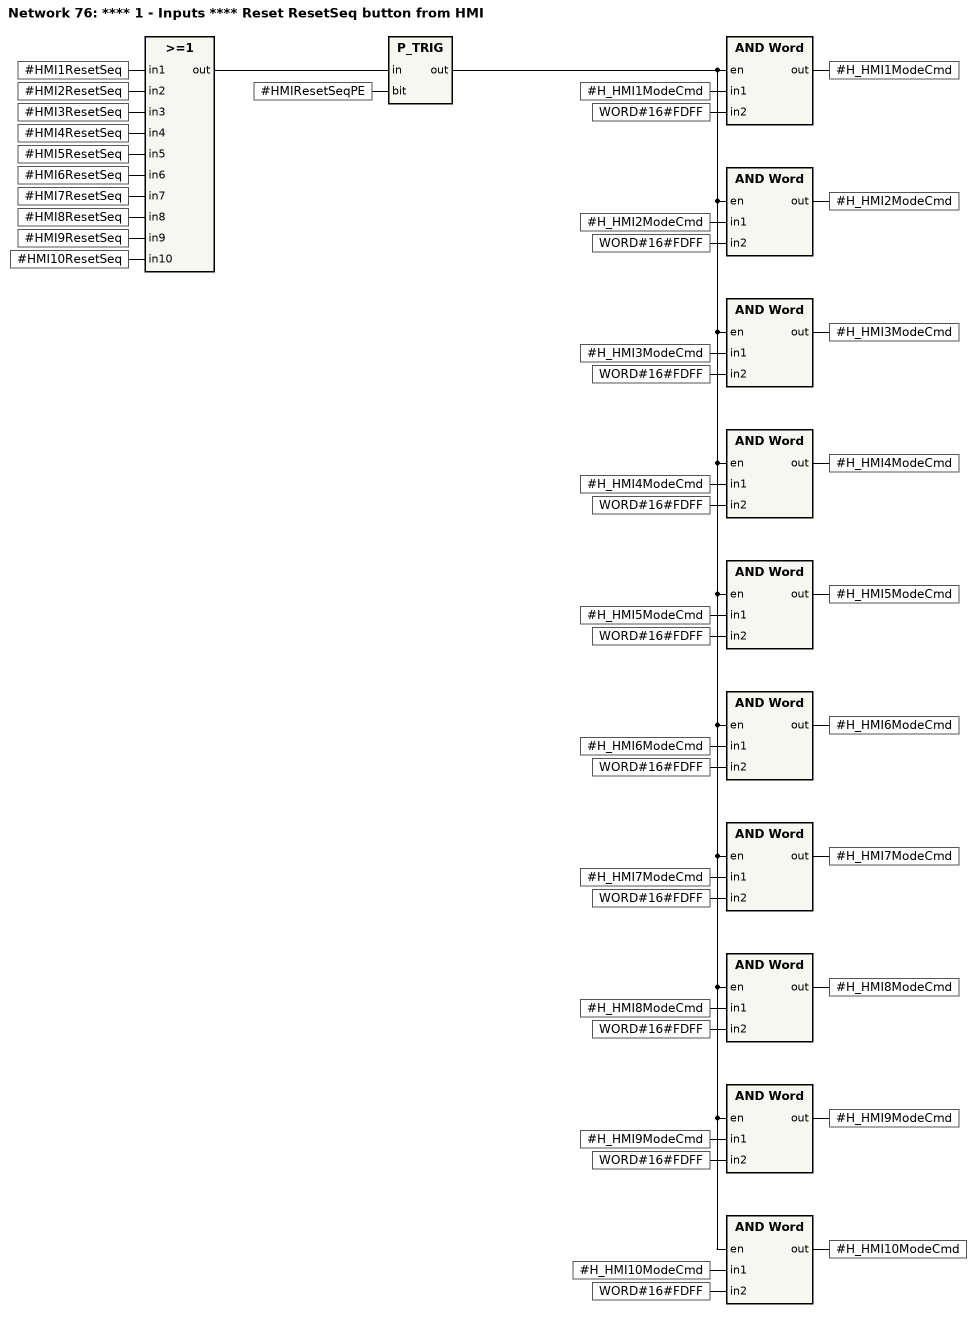
   #_w1 := #HMI1ResetSeq OR #HMI2ResetSeq OR #HMI3ResetSeq OR #HMI4ResetSeq OR #HMI5ResetSeq OR #HMI6ResetSeq OR #HMI7ResetSeq OR #HMI8ResetSeq OR #HMI9ResetSeq OR #HMI10ResetSeq;
   #_w2 := #_w1 AND NOT #HMIResetSeqPE;   // rising edge
   #HMIResetSeqPE := #_w1;
   IF #_w2 THEN
       #H_HMI1ModeCmd := #H_HMI1ModeCmd AND WORD#16#FDFF;
       #H_HMI2ModeCmd := #H_HMI2ModeCmd AND WORD#16#FDFF;
       #H_HMI3ModeCmd := #H_HMI3ModeCmd AND WORD#16#FDFF;
       #H_HMI4ModeCmd := #H_HMI4ModeCmd AND WORD#16#FDFF;
       #H_HMI5ModeCmd := #H_HMI5ModeCmd AND WORD#16#FDFF;
       #H_HMI6ModeCmd := #H_HMI6ModeCmd AND WORD#16#FDFF;
       #H_HMI7ModeCmd := #H_HMI7ModeCmd AND WORD#16#FDFF;
       #H_HMI8ModeCmd := #H_HMI8ModeCmd AND WORD#16#FDFF;
       #H_HMI9ModeCmd := #H_HMI9ModeCmd AND WORD#16#FDFF;
       #H_HMI10ModeCmd := #H_HMI10ModeCmd AND WORD#16#FDFF;
   END_IF;
END_REGION

REGION Network 77: **** 1 - Inputs **** Reset LockManual button from HMI
   // Reset LockManual button from HMI
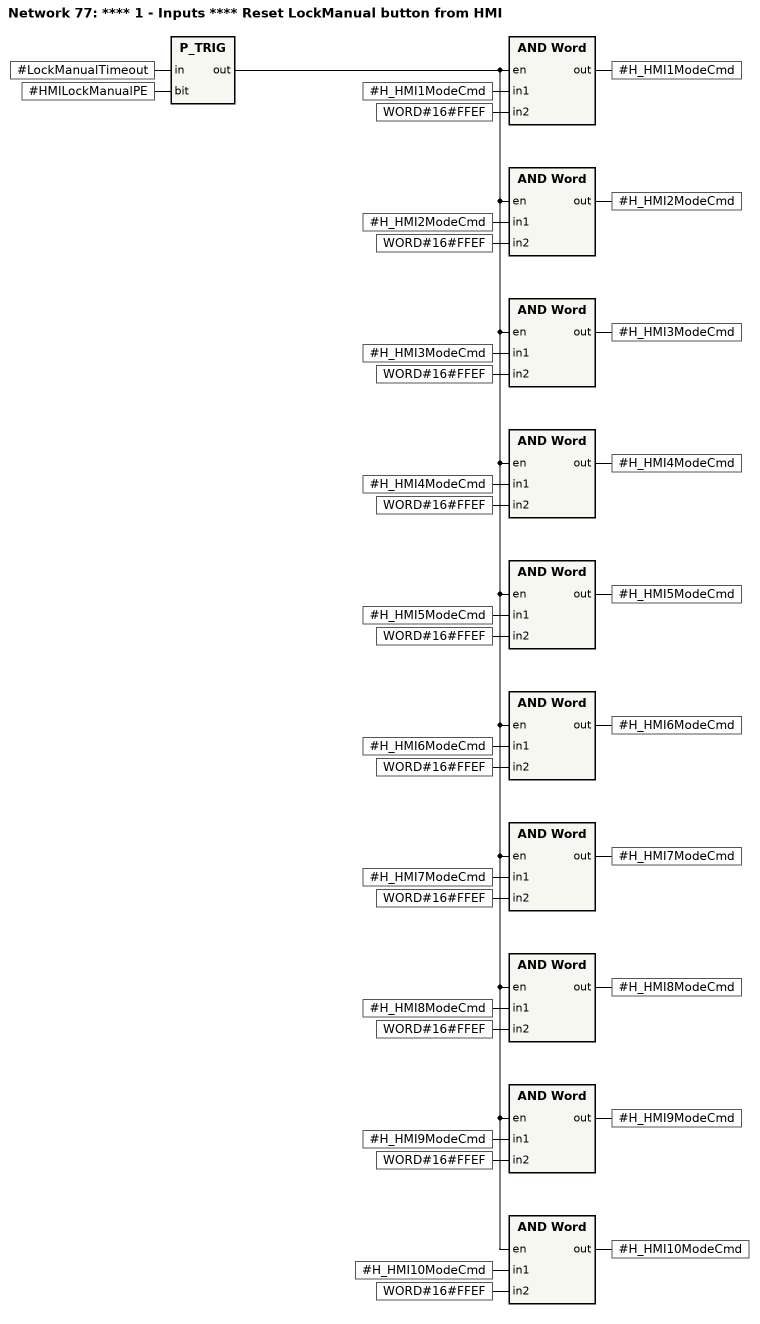
   #_w1 := #LockManualTimeout AND NOT #HMILockManualPE;   // rising edge
   #HMILockManualPE := #LockManualTimeout;
   IF #_w1 THEN
       #H_HMI1ModeCmd := #H_HMI1ModeCmd AND WORD#16#FFEF;
       #H_HMI2ModeCmd := #H_HMI2ModeCmd AND WORD#16#FFEF;
       #H_HMI3ModeCmd := #H_HMI3ModeCmd AND WORD#16#FFEF;
       #H_HMI4ModeCmd := #H_HMI4ModeCmd AND WORD#16#FFEF;
       #H_HMI5ModeCmd := #H_HMI5ModeCmd AND WORD#16#FFEF;
       #H_HMI6ModeCmd := #H_HMI6ModeCmd AND WORD#16#FFEF;
       #H_HMI7ModeCmd := #H_HMI7ModeCmd AND WORD#16#FFEF;
       #H_HMI8ModeCmd := #H_HMI8ModeCmd AND WORD#16#FFEF;
       #H_HMI9ModeCmd := #H_HMI9ModeCmd AND WORD#16#FFEF;
       #H_HMI10ModeCmd := #H_HMI10ModeCmd AND WORD#16#FFEF;
   END_IF;
END_REGION

REGION Network 78: **** 1 - Inputs **** Set Auto select on HMI-1 if plc go from STOP to RUN
   // Set Auto select on HMI-1 with the first scan
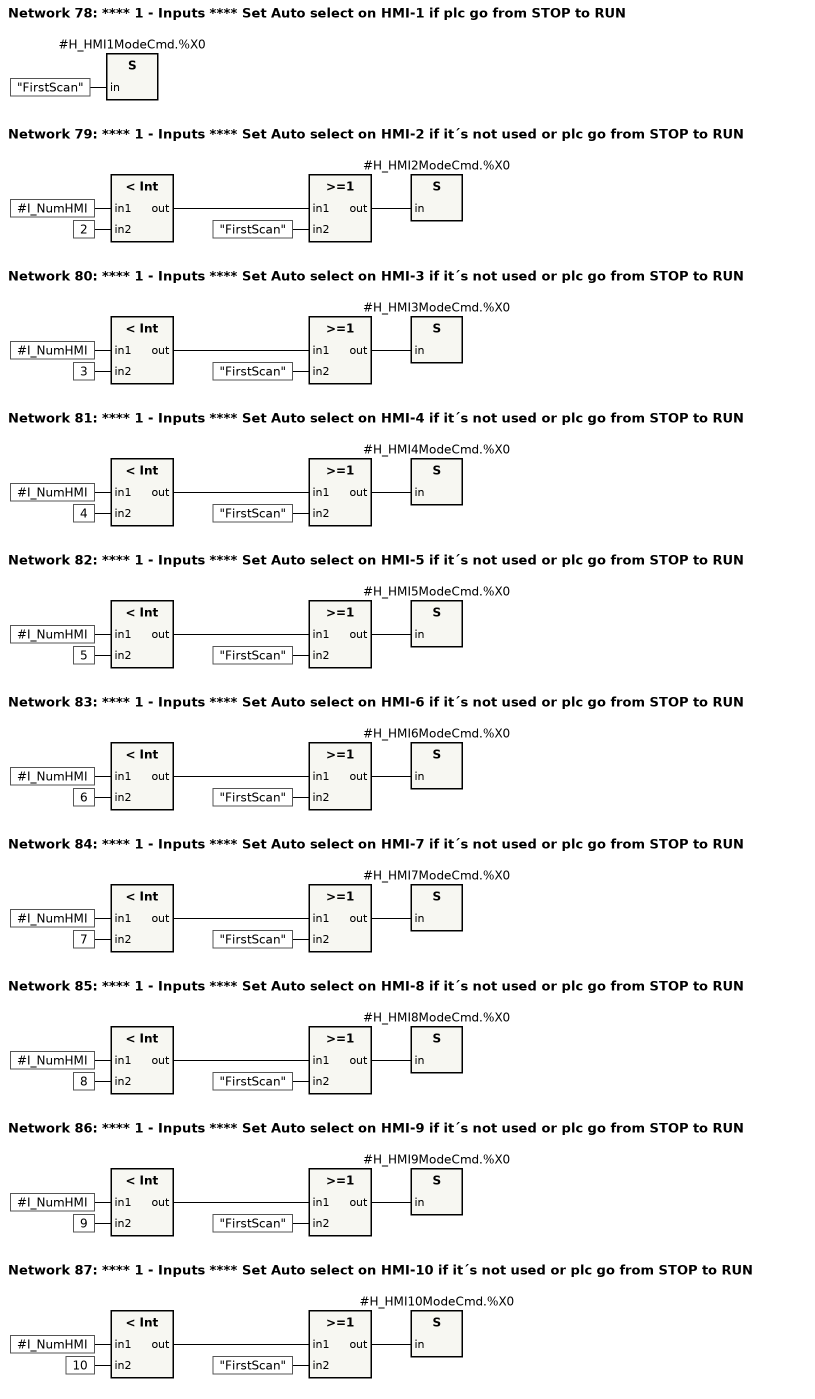
   IF "FirstScan" THEN #H_HMI1ModeCmd.%X0 := TRUE; END_IF;
END_REGION

REGION Network 79: **** 1 - Inputs **** Set Auto select on HMI-2 if it´s not used or plc go from STOP to RUN
   // Set Auto select on HMI-2 if it´s not used
   IF (#I_NumHMI < 2) OR "FirstScan" THEN #H_HMI2ModeCmd.%X0 := TRUE; END_IF;
END_REGION

REGION Network 80: **** 1 - Inputs **** Set Auto select on HMI-3 if it´s not used or plc go from STOP to RUN
   // Set Auto select on HMI-3 if it´s not used
   IF (#I_NumHMI < 3) OR "FirstScan" THEN #H_HMI3ModeCmd.%X0 := TRUE; END_IF;
END_REGION

REGION Network 81: **** 1 - Inputs **** Set Auto select on HMI-4 if it´s not used or plc go from STOP to RUN
   // Set Auto select on HMI-4 if it´s not used
   IF (#I_NumHMI < 4) OR "FirstScan" THEN #H_HMI4ModeCmd.%X0 := TRUE; END_IF;
END_REGION

REGION Network 82: **** 1 - Inputs **** Set Auto select on HMI-5 if it´s not used or plc go from STOP to RUN
   // Set Auto select on HMI-5 if it´s not used
   IF (#I_NumHMI < 5) OR "FirstScan" THEN #H_HMI5ModeCmd.%X0 := TRUE; END_IF;
END_REGION

REGION Network 83: **** 1 - Inputs **** Set Auto select on HMI-6 if it´s not used or plc go from STOP to RUN
   // Set Auto select on HMI-6 if it´s not used
   IF (#I_NumHMI < 6) OR "FirstScan" THEN #H_HMI6ModeCmd.%X0 := TRUE; END_IF;
END_REGION

REGION Network 84: **** 1 - Inputs **** Set Auto select on HMI-7 if it´s not used or plc go from STOP to RUN
   // Set Auto select on HMI-7 if it´s not used
   IF (#I_NumHMI < 7) OR "FirstScan" THEN #H_HMI7ModeCmd.%X0 := TRUE; END_IF;
END_REGION

REGION Network 85: **** 1 - Inputs **** Set Auto select on HMI-8 if it´s not used or plc go from STOP to RUN
   // Set Auto select on HMI-8 if it´s not used
   IF (#I_NumHMI < 8) OR "FirstScan" THEN #H_HMI8ModeCmd.%X0 := TRUE; END_IF;
END_REGION

REGION Network 86: **** 1 - Inputs **** Set Auto select on HMI-9 if it´s not used or plc go from STOP to RUN
   // Set Auto select on HMI-9 if it´s not used
   IF (#I_NumHMI < 9) OR "FirstScan" THEN #H_HMI9ModeCmd.%X0 := TRUE; END_IF;
END_REGION

REGION Network 87: **** 1 - Inputs **** Set Auto select on HMI-10 if it´s not used or plc go from STOP to RUN
   // Set Auto select on HMI-10 if it´s not used
   IF (#I_NumHMI < 10) OR "FirstScan" THEN #H_HMI10ModeCmd.%X0 := TRUE; END_IF;
END_REGION

REGION Network 88: **** 4.3 - Machine Status - Operator Sel **** Forced manual is selected on the active HMI
   // Forced manual is selected on the active HMI
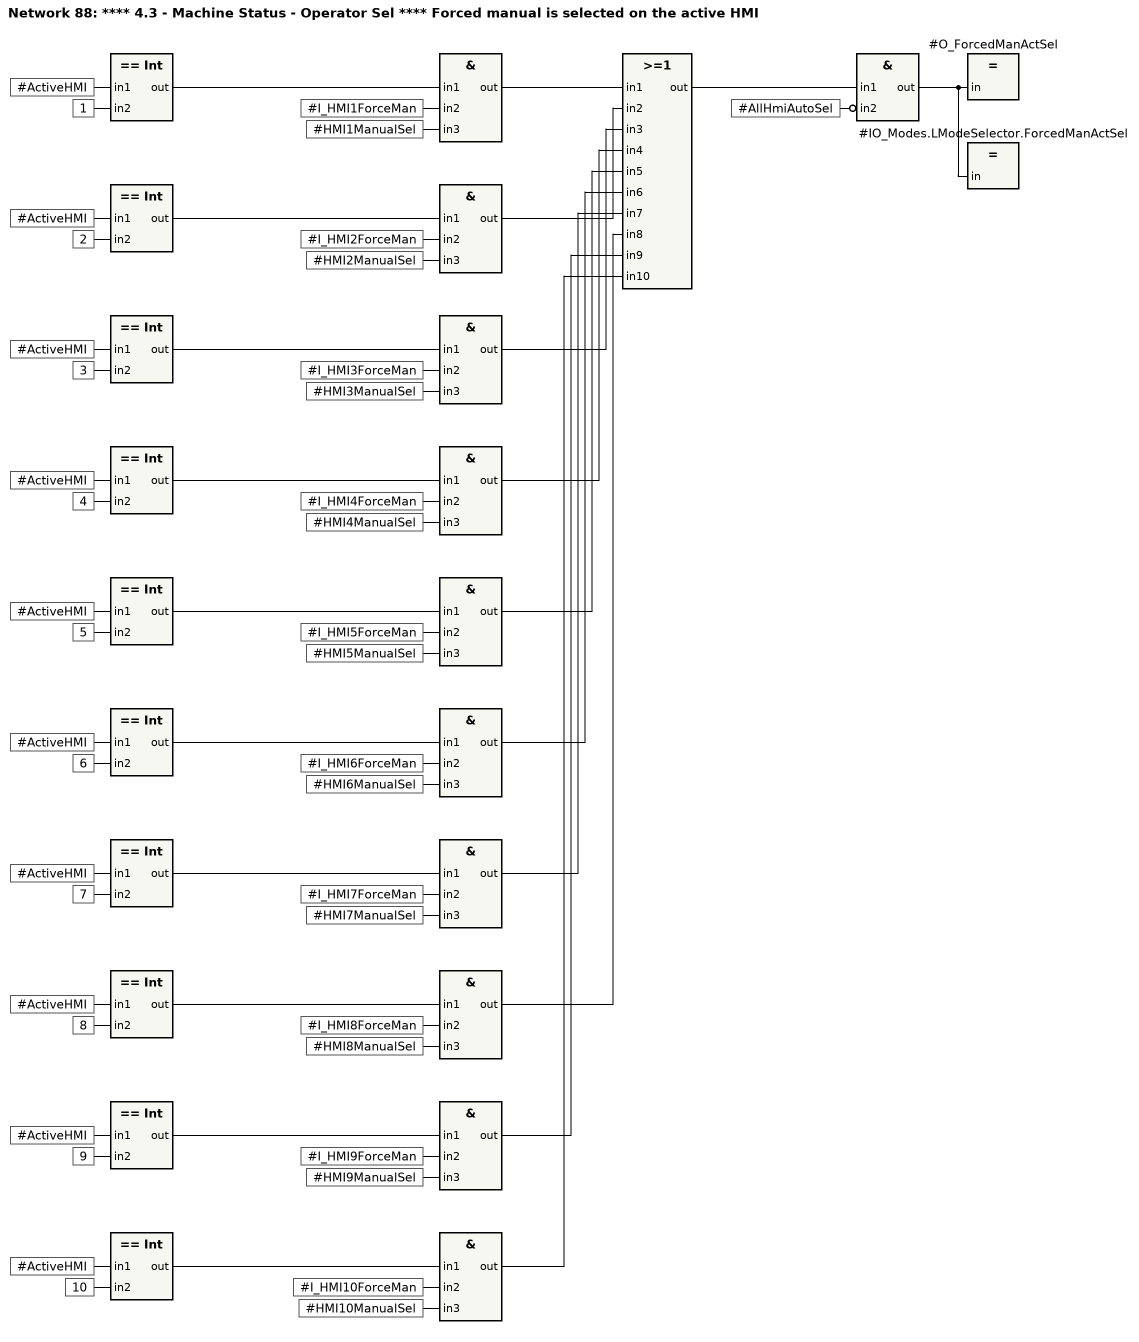
   #O_ForcedManActSel := (((#ActiveHMI = 1) AND #I_HMI1ForceMan AND #HMI1ManualSel) OR ((#ActiveHMI = 2) AND #I_HMI2ForceMan AND #HMI2ManualSel) OR ((#ActiveHMI = 3) AND #I_HMI3ForceMan AND #HMI3ManualSel) OR ((#ActiveHMI = 4) AND #I_HMI4ForceMan AND #HMI4ManualSel) OR ((#ActiveHMI = 5) AND #I_HMI5ForceMan AND #HMI5ManualSel) OR ((#ActiveHMI = 6) AND #I_HMI6ForceMan AND #HMI6ManualSel) OR ((#ActiveHMI = 7) AND #I_HMI7ForceMan AND #HMI7ManualSel) OR ((#ActiveHMI = 8) AND #I_HMI8ForceMan AND #HMI8ManualSel) OR ((#ActiveHMI = 9) AND #I_HMI9ForceMan AND #HMI9ManualSel) OR ((#ActiveHMI = 10) AND #I_HMI10ForceMan AND #HMI10ManualSel)) AND NOT #AllHmiAutoSel;
   #IO_Modes.LModeSelector.ForcedManActSel := #O_ForcedManActSel;
END_REGION

REGION Network 89: **** 4.3 - Machine Status - Operator Sel **** Set pushbutton is selected on the active HMI
   // Set pushbutton is selected on the active HMI
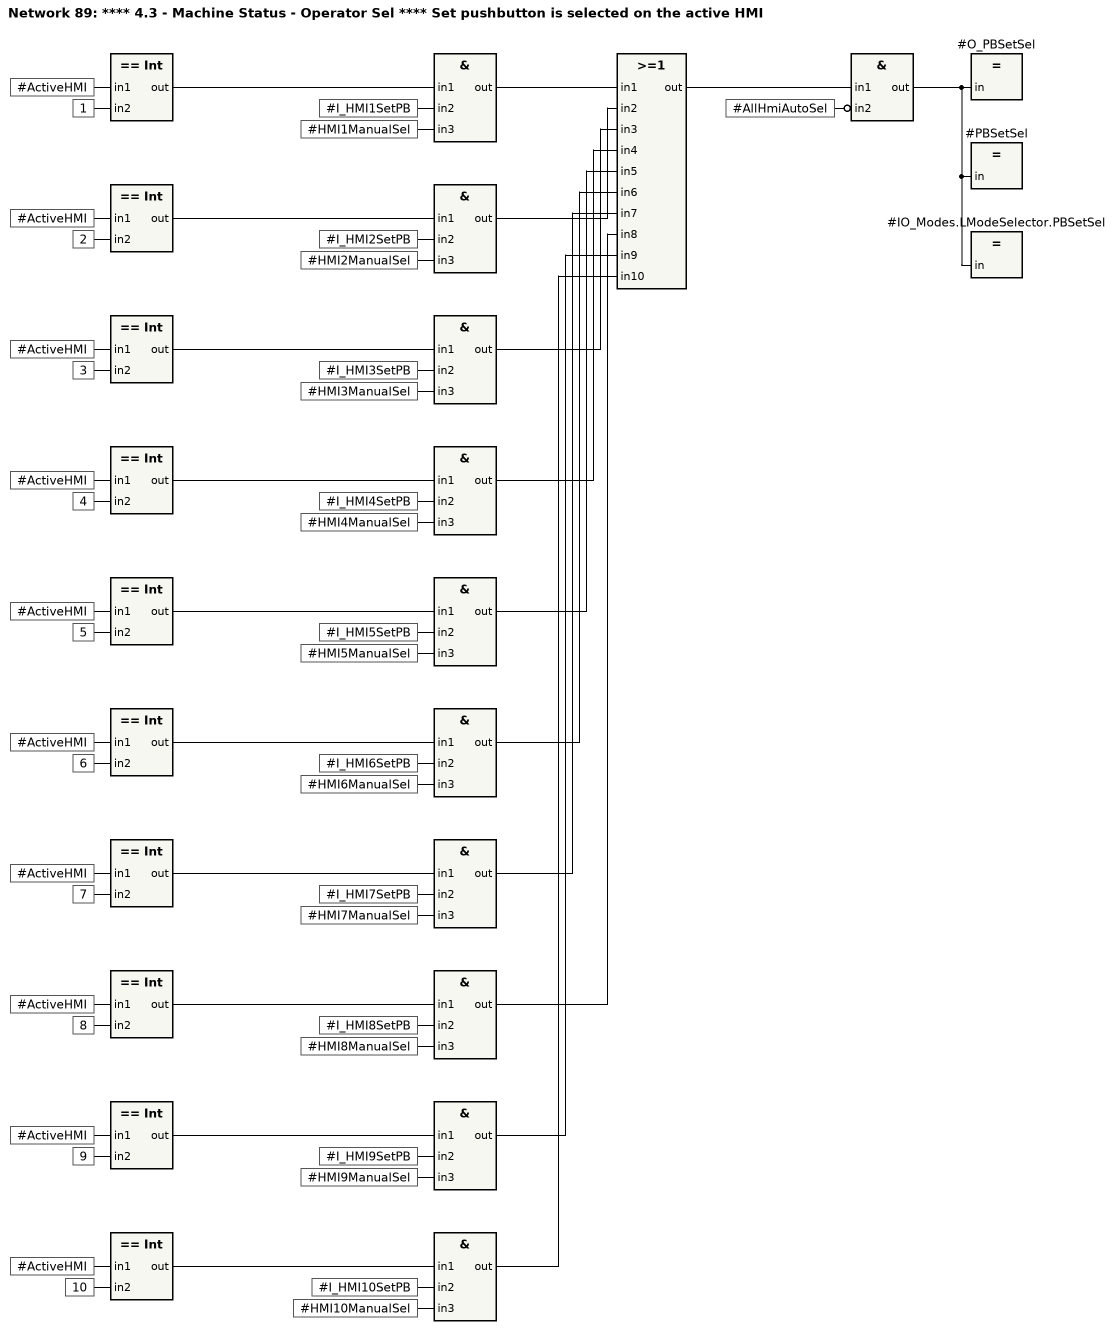
   #O_PBSetSel := (((#ActiveHMI = 1) AND #I_HMI1SetPB AND #HMI1ManualSel) OR ((#ActiveHMI = 2) AND #I_HMI2SetPB AND #HMI2ManualSel) OR ((#ActiveHMI = 3) AND #I_HMI3SetPB AND #HMI3ManualSel) OR ((#ActiveHMI = 4) AND #I_HMI4SetPB AND #HMI4ManualSel) OR ((#ActiveHMI = 5) AND #I_HMI5SetPB AND #HMI5ManualSel) OR ((#ActiveHMI = 6) AND #I_HMI6SetPB AND #HMI6ManualSel) OR ((#ActiveHMI = 7) AND #I_HMI7SetPB AND #HMI7ManualSel) OR ((#ActiveHMI = 8) AND #I_HMI8SetPB AND #HMI8ManualSel) OR ((#ActiveHMI = 9) AND #I_HMI9SetPB AND #HMI9ManualSel) OR ((#ActiveHMI = 10) AND #I_HMI10SetPB AND #HMI10ManualSel)) AND NOT #AllHmiAutoSel;
   #PBSetSel := #O_PBSetSel;
   #IO_Modes.LModeSelector.PBSetSel := #O_PBSetSel;
END_REGION

REGION Network 90: **** 4.3 - Machine Status - Operator Sel **** Reset pushbutton is selected on the active HMI
   // Reset pushbutton is selected on the active HMI
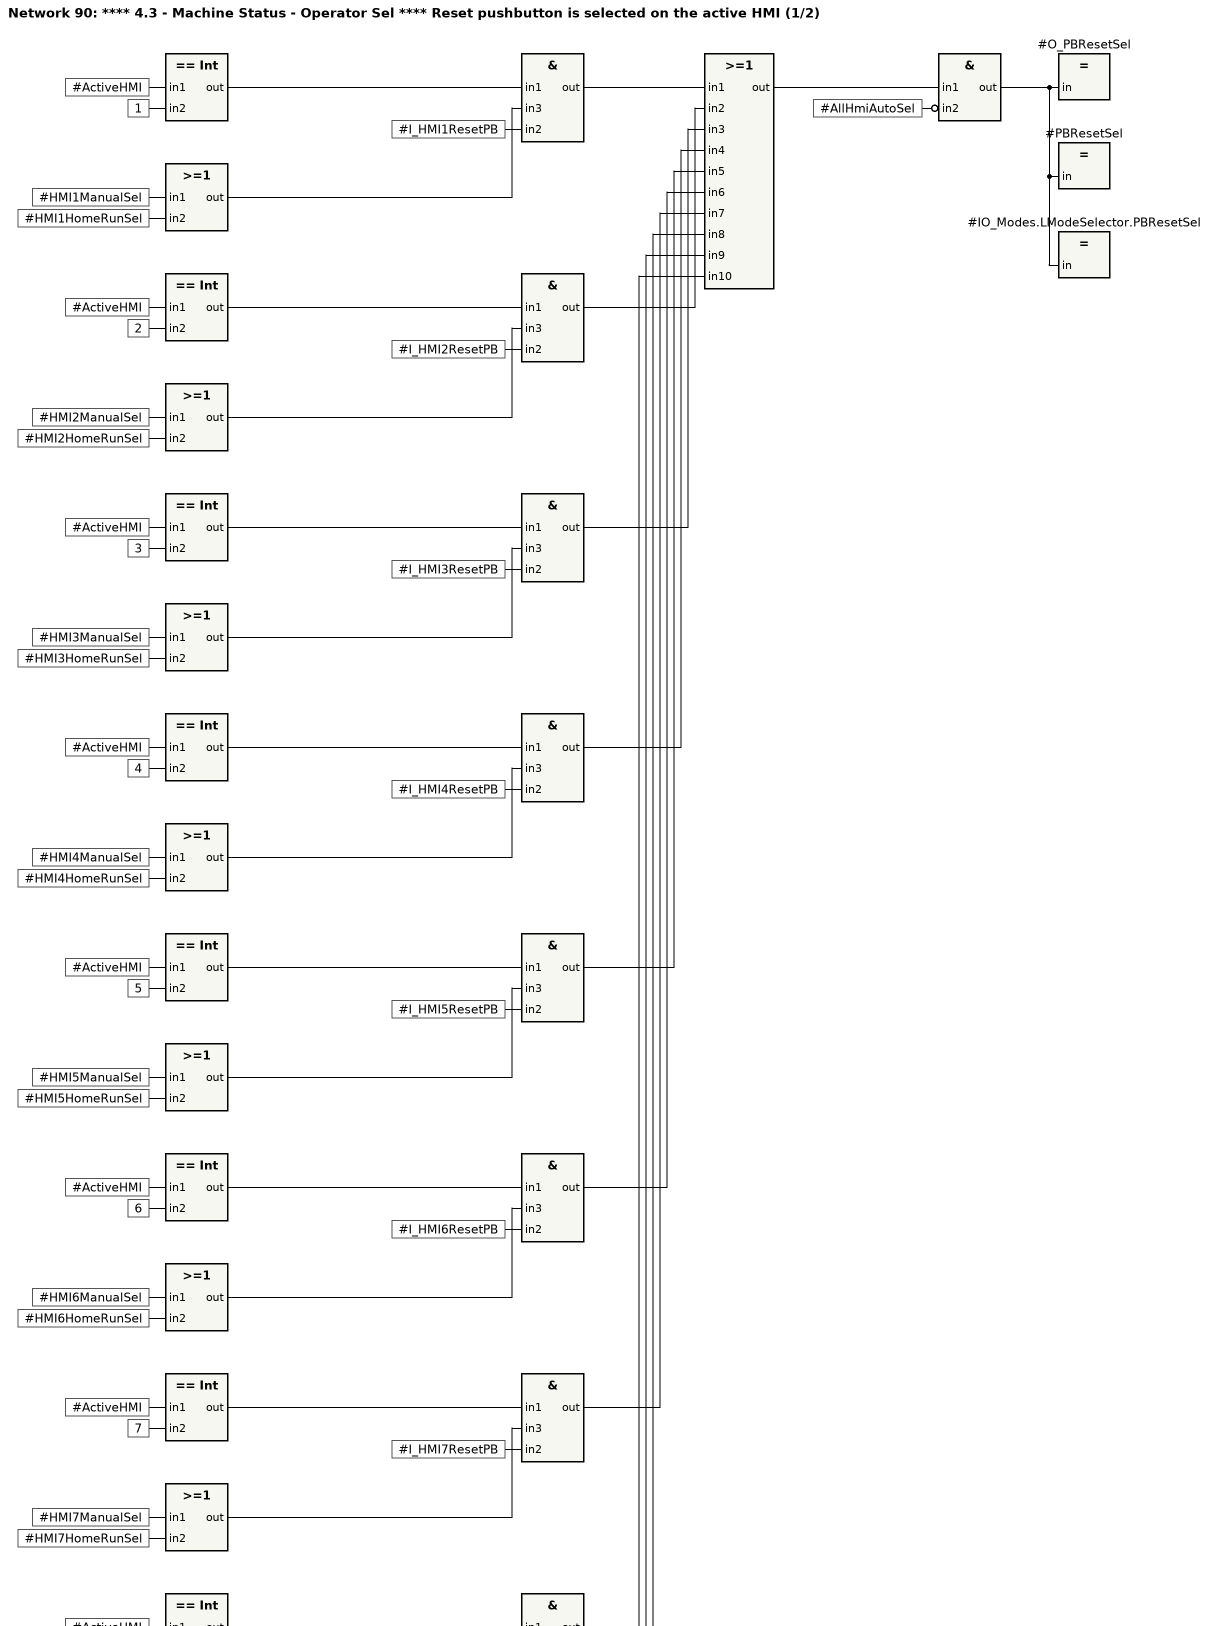
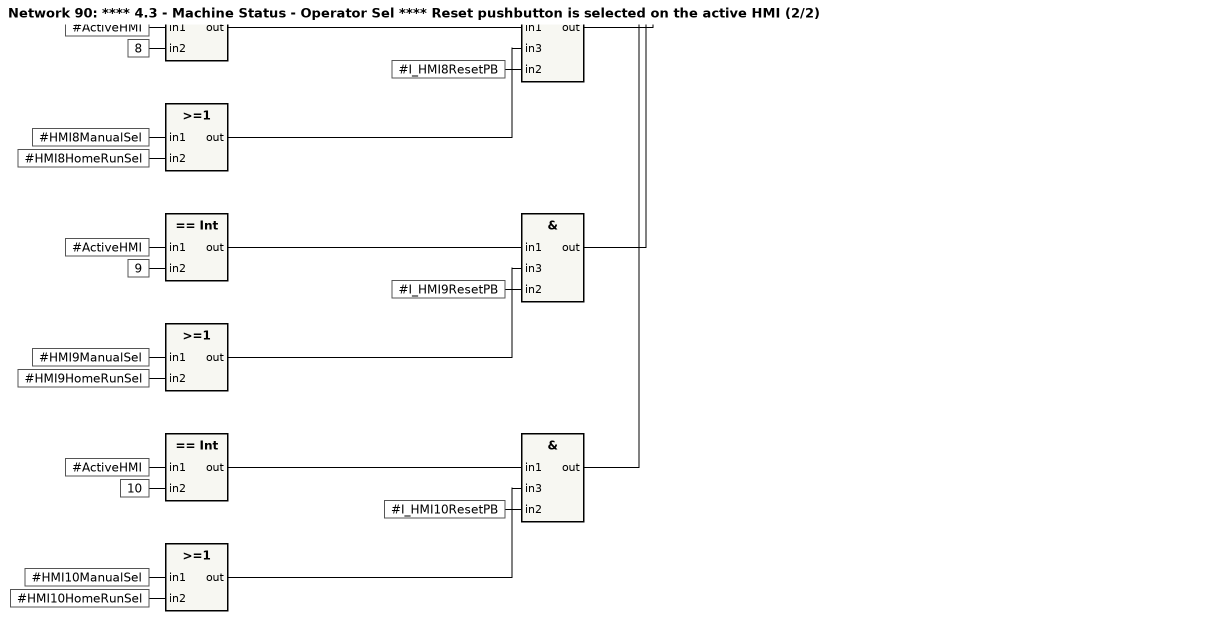
   #O_PBResetSel := (((#ActiveHMI = 1) AND (#HMI1ManualSel OR #HMI1HomeRunSel) AND #I_HMI1ResetPB) OR ((#ActiveHMI = 2) AND (#HMI2ManualSel OR #HMI2HomeRunSel) AND #I_HMI2ResetPB) OR ((#ActiveHMI = 3) AND (#HMI3ManualSel OR #HMI3HomeRunSel) AND #I_HMI3ResetPB) OR ((#ActiveHMI = 4) AND (#HMI4ManualSel OR #HMI4HomeRunSel) AND #I_HMI4ResetPB) OR ((#ActiveHMI = 5) AND (#HMI5ManualSel OR #HMI5HomeRunSel) AND #I_HMI5ResetPB) OR ((#ActiveHMI = 6) AND (#HMI6ManualSel OR #HMI6HomeRunSel) AND #I_HMI6ResetPB) OR ((#ActiveHMI = 7) AND (#HMI7ManualSel OR #HMI7HomeRunSel) AND #I_HMI7ResetPB) OR ((#ActiveHMI = 8) AND (#HMI8ManualSel OR #HMI8HomeRunSel) AND #I_HMI8ResetPB) OR ((#ActiveHMI = 9) AND (#HMI9ManualSel OR #HMI9HomeRunSel) AND #I_HMI9ResetPB) OR ((#ActiveHMI = 10) AND (#HMI10ManualSel OR #HMI10HomeRunSel) AND #I_HMI10ResetPB)) AND NOT #AllHmiAutoSel;
   #PBResetSel := #O_PBResetSel;
   #IO_Modes.LModeSelector.PBResetSel := #O_PBResetSel;
END_REGION

REGION Network 91: **** 4.3 - Machine Status - Operator Sel **** Homerun Redo is selected
   // Homerun Redo is selected
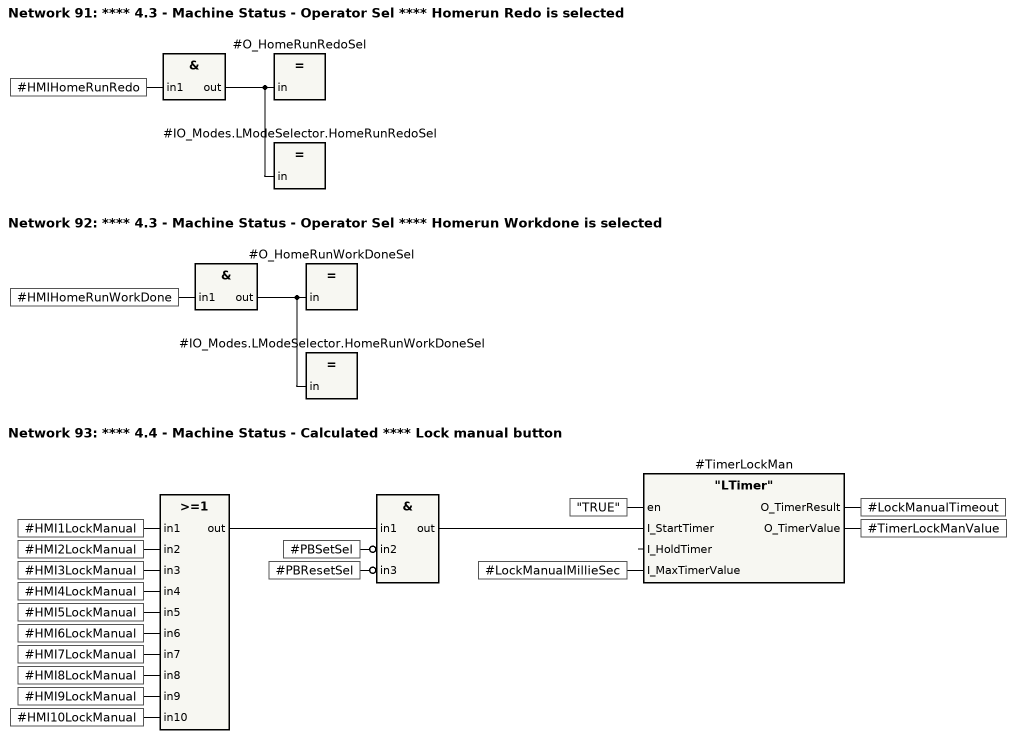
   #O_HomeRunRedoSel := #HMIHomeRunRedo;
   #IO_Modes.LModeSelector.HomeRunRedoSel := #HMIHomeRunRedo;
END_REGION

REGION Network 92: **** 4.3 - Machine Status - Operator Sel **** Homerun Workdone is selected
   // Homerun Workdone is selected
   #O_HomeRunWorkDoneSel := #HMIHomeRunWorkDone;
   #IO_Modes.LModeSelector.HomeRunWorkDoneSel := #HMIHomeRunWorkDone;
END_REGION

REGION Network 93: **** 4.4 - Machine Status - Calculated **** Lock manual button
   // Lock manual button
   IF "TRUE" THEN
       #TimerLockMan(I_StartTimer := (#HMI1LockManual OR #HMI2LockManual OR #HMI3LockManual OR #HMI4LockManual OR #HMI5LockManual OR #HMI6LockManual OR #HMI7LockManual OR #HMI8LockManual OR #HMI9LockManual OR #HMI10LockManual) AND NOT #PBSetSel AND NOT #PBResetSel,   // "LTimer"
                     I_MaxTimerValue := #LockManualMillieSec,
                     O_TimerResult => #LockManualTimeout,
                     O_TimerValue => #TimerLockManValue);
   END_IF;
END_REGION

REGION Network 94: **** 4.5 - Machine Status - Modes **** Auto is selected on all HMI
   // Auto is selected on all HMI
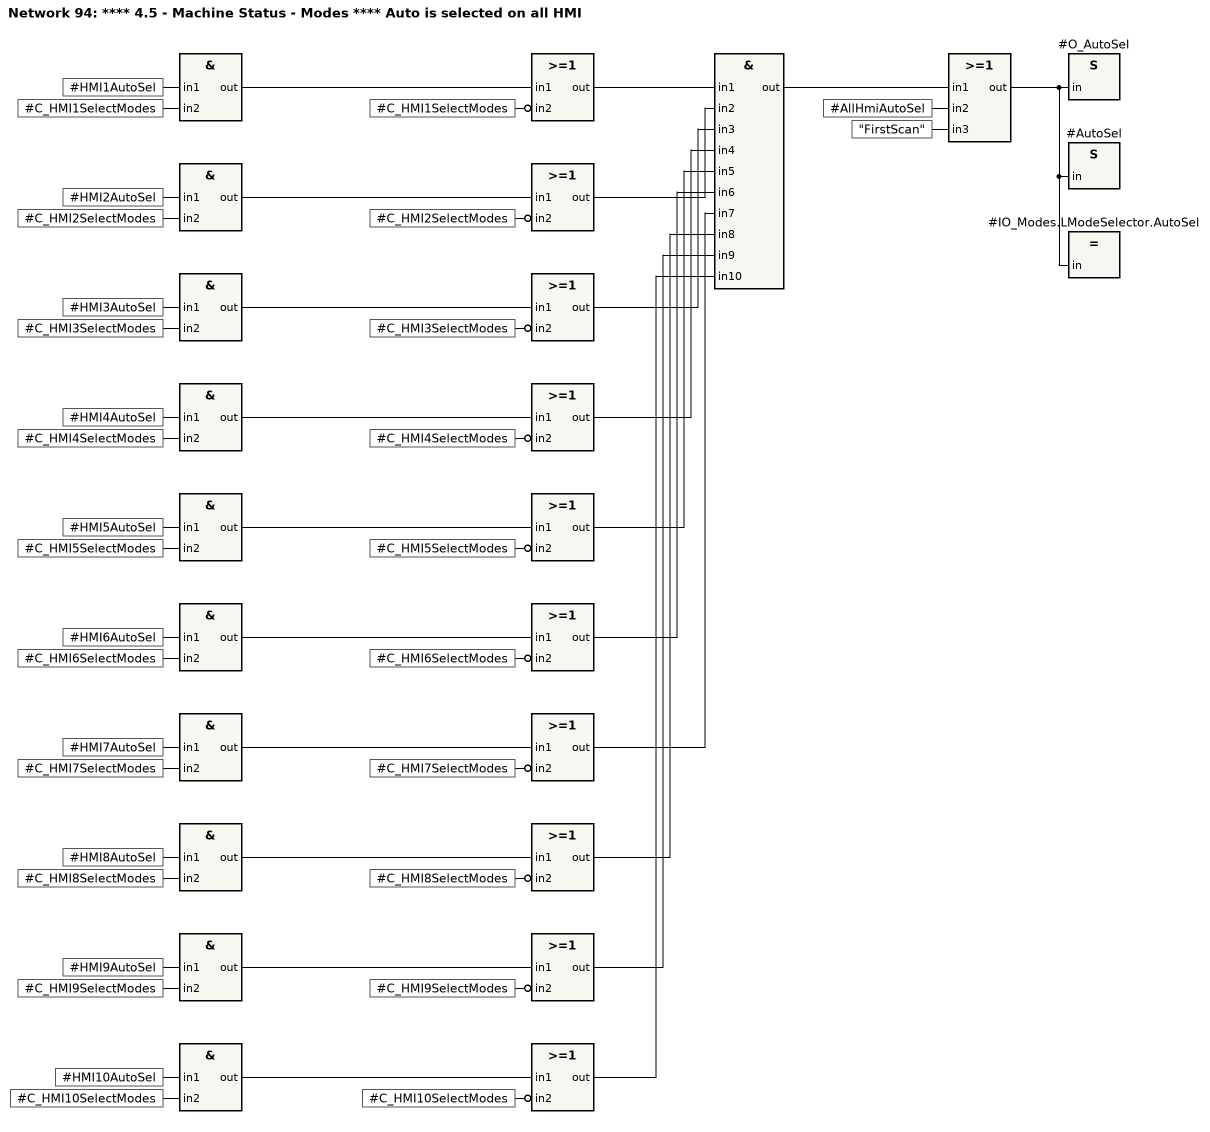
   #_w1 := (((#HMI1AutoSel AND #C_HMI1SelectModes) OR NOT #C_HMI1SelectModes) AND ((#HMI2AutoSel AND #C_HMI2SelectModes) OR NOT #C_HMI2SelectModes) AND ((#HMI3AutoSel AND #C_HMI3SelectModes) OR NOT #C_HMI3SelectModes) AND ((#HMI4AutoSel AND #C_HMI4SelectModes) OR NOT #C_HMI4SelectModes) AND ((#HMI5AutoSel AND #C_HMI5SelectModes) OR NOT #C_HMI5SelectModes) AND ((#HMI6AutoSel AND #C_HMI6SelectModes) OR NOT #C_HMI6SelectModes) AND ((#HMI7AutoSel AND #C_HMI7SelectModes) OR NOT #C_HMI7SelectModes) AND ((#HMI8AutoSel AND #C_HMI8SelectModes) OR NOT #C_HMI8SelectModes) AND ((#HMI9AutoSel AND #C_HMI9SelectModes) OR NOT #C_HMI9SelectModes) AND ((#HMI10AutoSel AND #C_HMI10SelectModes) OR NOT #C_HMI10SelectModes)) OR #AllHmiAutoSel OR "FirstScan";
   IF #_w1 THEN
       #O_AutoSel := TRUE;
       #AutoSel := TRUE;
   END_IF;
   #IO_Modes.LModeSelector.AutoSel := #_w1;
END_REGION

REGION Network 95: **** 4.5 - Machine Status - Modes **** Reset Auto is selected on all HMI
   // Reset Auto is selected on all HMI
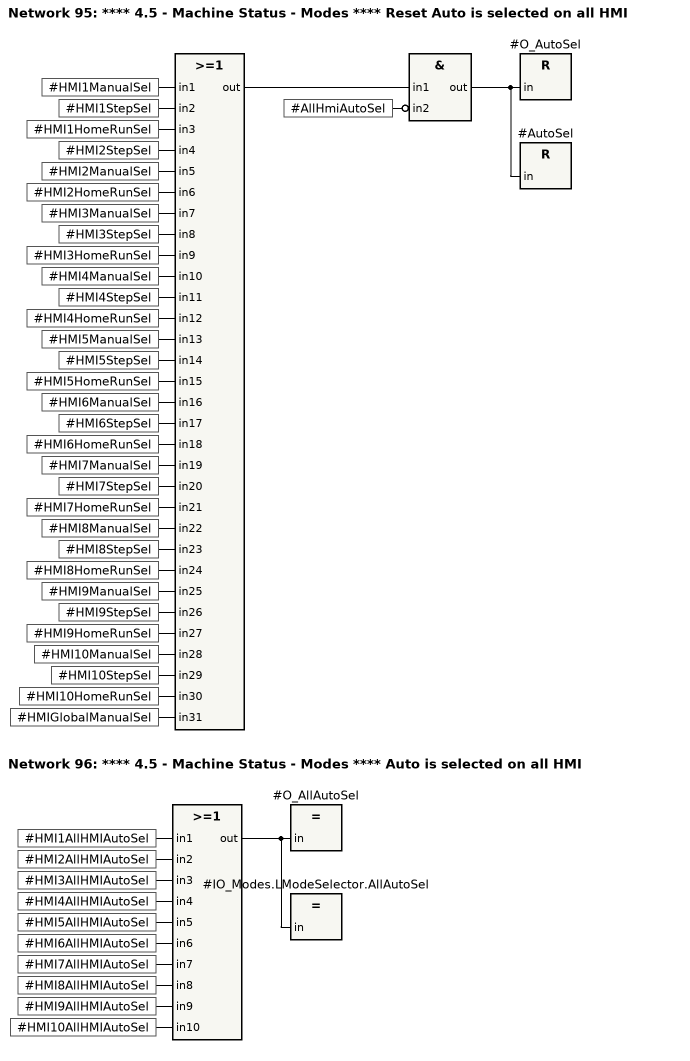
   IF (#HMI1ManualSel OR #HMI1StepSel OR #HMI1HomeRunSel OR #HMI2StepSel OR #HMI2ManualSel OR #HMI2HomeRunSel OR #HMI3ManualSel OR #HMI3StepSel OR #HMI3HomeRunSel OR #HMI4ManualSel OR #HMI4StepSel OR #HMI4HomeRunSel OR #HMI5ManualSel OR #HMI5StepSel OR #HMI5HomeRunSel OR #HMI6ManualSel OR #HMI6StepSel OR #HMI6HomeRunSel OR #HMI7ManualSel OR #HMI7StepSel OR #HMI7HomeRunSel OR #HMI8ManualSel OR #HMI8StepSel OR #HMI8HomeRunSel OR #HMI9ManualSel OR #HMI9StepSel OR #HMI9HomeRunSel OR #HMI10ManualSel OR #HMI10StepSel OR #HMI10HomeRunSel OR #HMIGlobalManualSel) AND NOT #AllHmiAutoSel THEN
       #O_AutoSel := FALSE;
       #AutoSel := FALSE;
   END_IF;
END_REGION

REGION Network 96: **** 4.5 - Machine Status - Modes **** Auto is selected on all HMI
   // Auto is selected on all HMI
   #O_AllAutoSel := #HMI1AllHMIAutoSel OR #HMI2AllHMIAutoSel OR #HMI3AllHMIAutoSel OR #HMI4AllHMIAutoSel OR #HMI5AllHMIAutoSel OR #HMI6AllHMIAutoSel OR #HMI7AllHMIAutoSel OR #HMI8AllHMIAutoSel OR #HMI9AllHMIAutoSel OR #HMI10AllHMIAutoSel;
   #IO_Modes.LModeSelector.AllAutoSel := #O_AllAutoSel;
END_REGION

REGION Network 97: **** 4.5 - Machine Status - Modes **** Step is selected on one HMI
   // Step is selected on one HMI
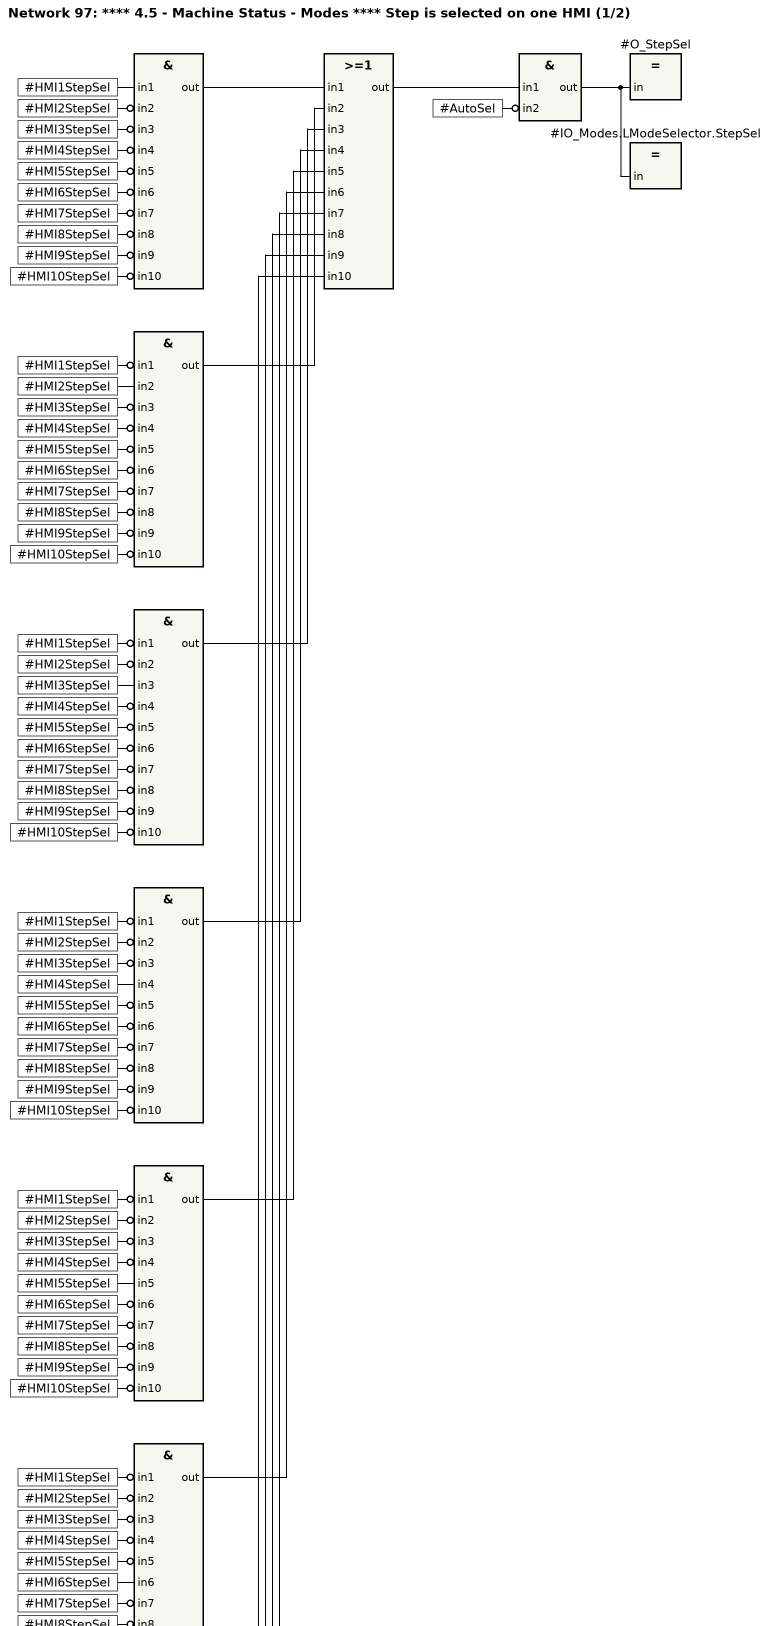
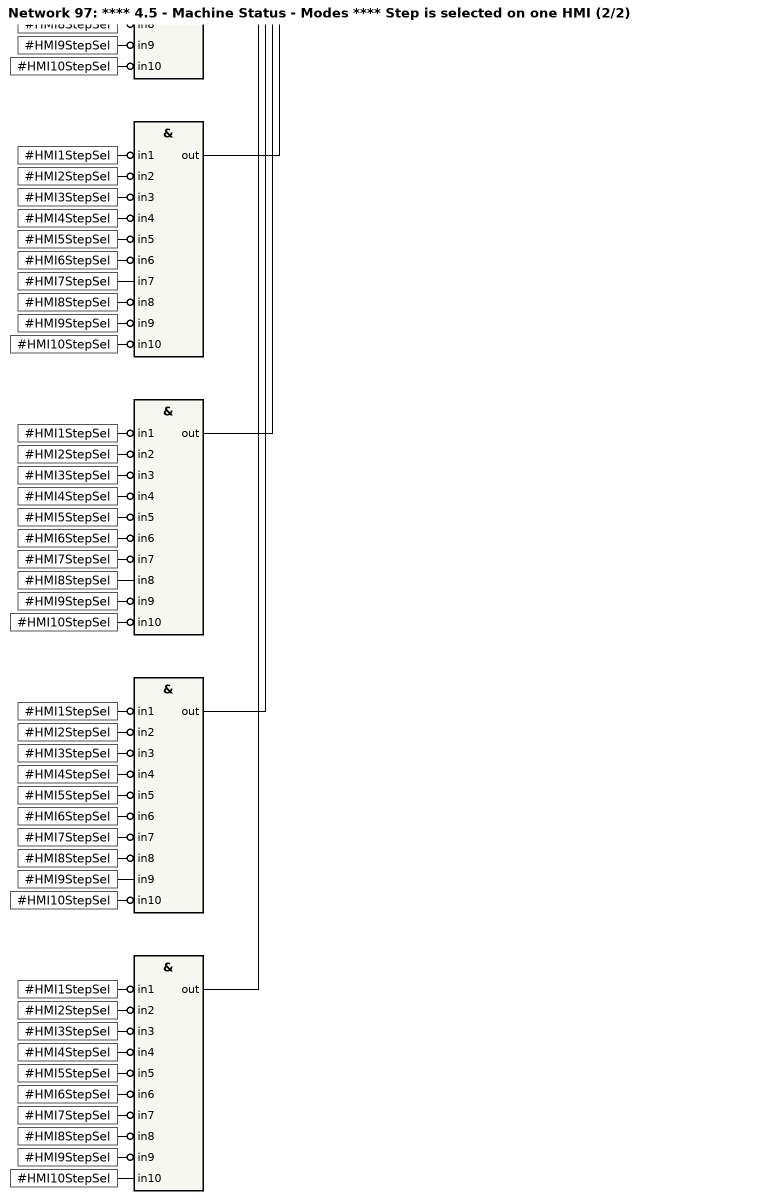
   #O_StepSel := ((#HMI1StepSel AND NOT #HMI2StepSel AND NOT #HMI3StepSel AND NOT #HMI4StepSel AND NOT #HMI5StepSel AND NOT #HMI6StepSel AND NOT #HMI7StepSel AND NOT #HMI8StepSel AND NOT #HMI9StepSel AND NOT #HMI10StepSel) OR (NOT #HMI1StepSel AND #HMI2StepSel AND NOT #HMI3StepSel AND NOT #HMI4StepSel AND NOT #HMI5StepSel AND NOT #HMI6StepSel AND NOT #HMI7StepSel AND NOT #HMI8StepSel AND NOT #HMI9StepSel AND NOT #HMI10StepSel) OR (NOT #HMI1StepSel AND NOT #HMI2StepSel AND #HMI3StepSel AND NOT #HMI4StepSel AND NOT #HMI5StepSel AND NOT #HMI6StepSel AND NOT #HMI7StepSel AND NOT #HMI8StepSel AND NOT #HMI9StepSel AND NOT #HMI10StepSel) OR (NOT #HMI1StepSel AND NOT #HMI2StepSel AND NOT #HMI3StepSel AND #HMI4StepSel AND NOT #HMI5StepSel AND NOT #HMI6StepSel AND NOT #HMI7StepSel AND NOT #HMI8StepSel AND NOT #HMI9StepSel AND NOT #HMI10StepSel) OR (NOT #HMI1StepSel AND NOT #HMI2StepSel AND NOT #HMI3StepSel AND NOT #HMI4StepSel AND #HMI5StepSel AND NOT #HMI6StepSel AND NOT #HMI7StepSel AND NOT #HMI8StepSel AND NOT #HMI9StepSel AND NOT #HMI10StepSel) OR (NOT #HMI1StepSel AND NOT #HMI2StepSel AND NOT #HMI3StepSel AND NOT #HMI4StepSel AND NOT #HMI5StepSel AND #HMI6StepSel AND NOT #HMI7StepSel AND NOT #HMI8StepSel AND NOT #HMI9StepSel AND NOT #HMI10StepSel) OR (NOT #HMI1StepSel AND NOT #HMI2StepSel AND NOT #HMI3StepSel AND NOT #HMI4StepSel AND NOT #HMI5StepSel AND NOT #HMI6StepSel AND #HMI7StepSel AND NOT #HMI8StepSel AND NOT #HMI9StepSel AND NOT #HMI10StepSel) OR (NOT #HMI1StepSel AND NOT #HMI2StepSel AND NOT #HMI3StepSel AND NOT #HMI4StepSel AND NOT #HMI5StepSel AND NOT #HMI6StepSel AND NOT #HMI7StepSel AND #HMI8StepSel AND NOT #HMI9StepSel AND NOT #HMI10StepSel) OR (NOT #HMI1StepSel AND NOT #HMI2StepSel AND NOT #HMI3StepSel AND NOT #HMI4StepSel AND NOT #HMI5StepSel AND NOT #HMI6StepSel AND NOT #HMI7StepSel AND NOT #HMI8StepSel AND #HMI9StepSel AND NOT #HMI10StepSel) OR (NOT #HMI1StepSel AND NOT #HMI2StepSel AND NOT #HMI3StepSel AND NOT #HMI4StepSel AND NOT #HMI5StepSel AND NOT #HMI6StepSel AND NOT #HMI7StepSel AND NOT #HMI8StepSel AND NOT #HMI9StepSel AND #HMI10StepSel)) AND NOT #AutoSel;
   #IO_Modes.LModeSelector.StepSel := #O_StepSel;
END_REGION

REGION Network 98: **** 4.5 - Machine Status - Modes **** Homerun is selected on one HMI
   // Homerun is selected on one HMI
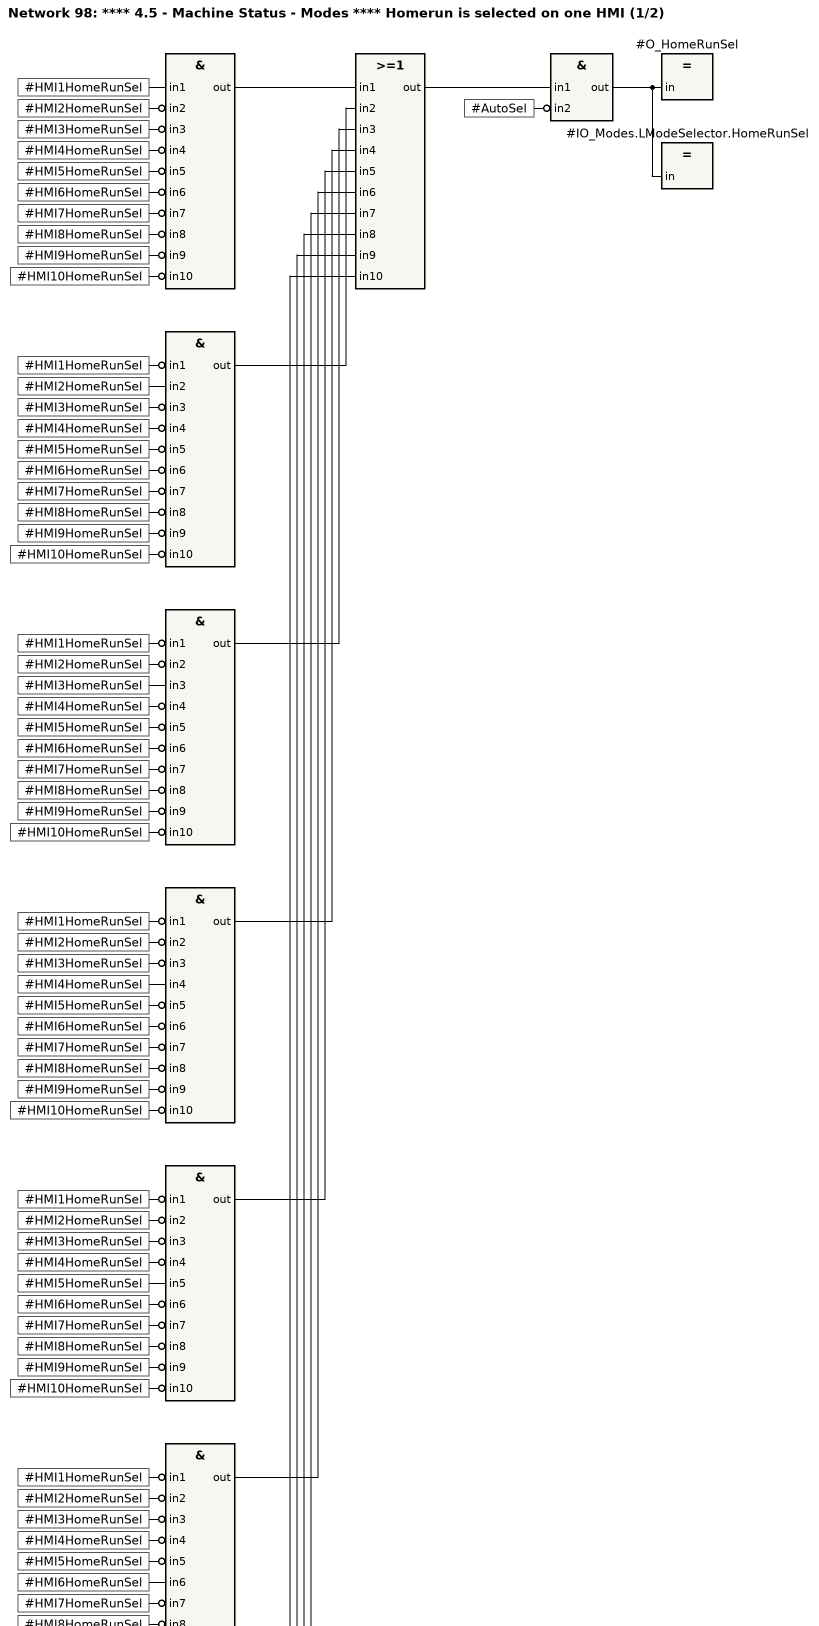
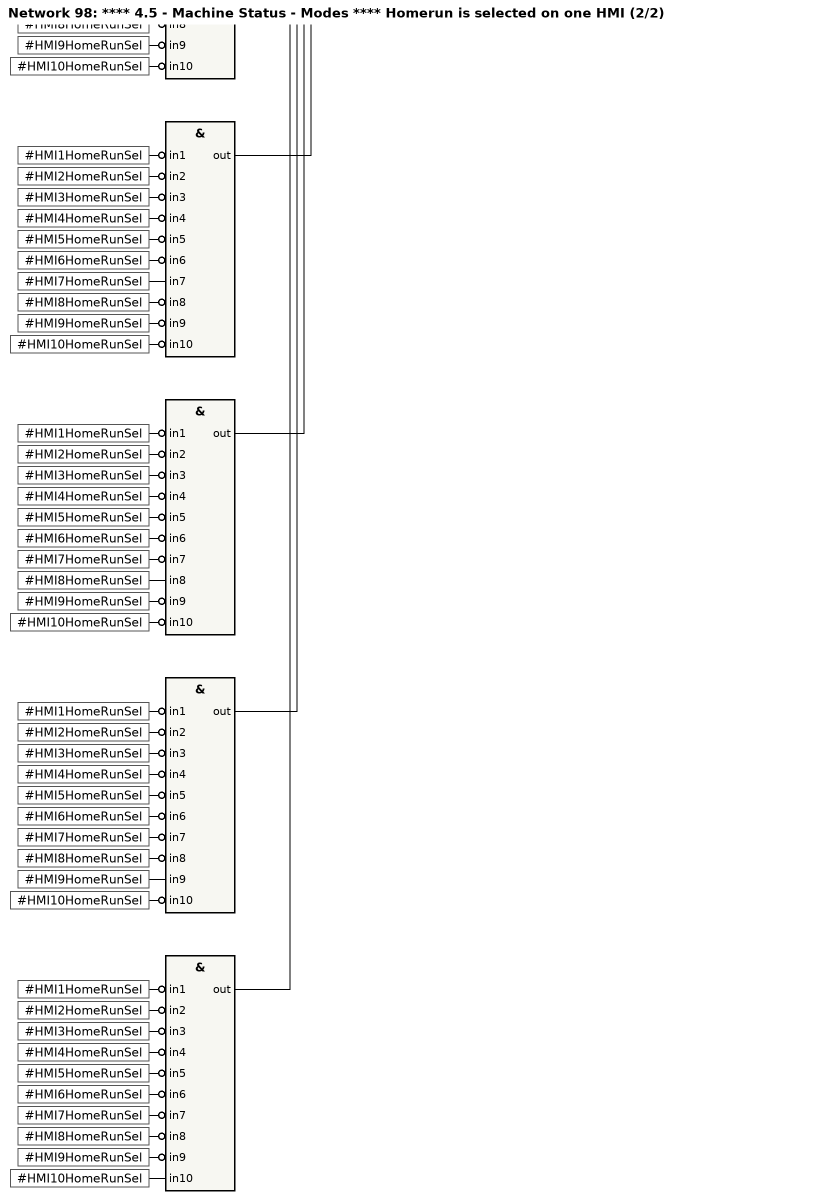
   #O_HomeRunSel := ((#HMI1HomeRunSel AND NOT #HMI2HomeRunSel AND NOT #HMI3HomeRunSel AND NOT #HMI4HomeRunSel AND NOT #HMI5HomeRunSel AND NOT #HMI6HomeRunSel AND NOT #HMI7HomeRunSel AND NOT #HMI8HomeRunSel AND NOT #HMI9HomeRunSel AND NOT #HMI10HomeRunSel) OR (NOT #HMI1HomeRunSel AND #HMI2HomeRunSel AND NOT #HMI3HomeRunSel AND NOT #HMI4HomeRunSel AND NOT #HMI5HomeRunSel AND NOT #HMI6HomeRunSel AND NOT #HMI7HomeRunSel AND NOT #HMI8HomeRunSel AND NOT #HMI9HomeRunSel AND NOT #HMI10HomeRunSel) OR (NOT #HMI1HomeRunSel AND NOT #HMI2HomeRunSel AND #HMI3HomeRunSel AND NOT #HMI4HomeRunSel AND NOT #HMI5HomeRunSel AND NOT #HMI6HomeRunSel AND NOT #HMI7HomeRunSel AND NOT #HMI8HomeRunSel AND NOT #HMI9HomeRunSel AND NOT #HMI10HomeRunSel) OR (NOT #HMI1HomeRunSel AND NOT #HMI2HomeRunSel AND NOT #HMI3HomeRunSel AND #HMI4HomeRunSel AND NOT #HMI5HomeRunSel AND NOT #HMI6HomeRunSel AND NOT #HMI7HomeRunSel AND NOT #HMI8HomeRunSel AND NOT #HMI9HomeRunSel AND NOT #HMI10HomeRunSel) OR (NOT #HMI1HomeRunSel AND NOT #HMI2HomeRunSel AND NOT #HMI3HomeRunSel AND NOT #HMI4HomeRunSel AND #HMI5HomeRunSel AND NOT #HMI6HomeRunSel AND NOT #HMI7HomeRunSel AND NOT #HMI8HomeRunSel AND NOT #HMI9HomeRunSel AND NOT #HMI10HomeRunSel) OR (NOT #HMI1HomeRunSel AND NOT #HMI2HomeRunSel AND NOT #HMI3HomeRunSel AND NOT #HMI4HomeRunSel AND NOT #HMI5HomeRunSel AND #HMI6HomeRunSel AND NOT #HMI7HomeRunSel AND NOT #HMI8HomeRunSel AND NOT #HMI9HomeRunSel AND NOT #HMI10HomeRunSel) OR (NOT #HMI1HomeRunSel AND NOT #HMI2HomeRunSel AND NOT #HMI3HomeRunSel AND NOT #HMI4HomeRunSel AND NOT #HMI5HomeRunSel AND NOT #HMI6HomeRunSel AND #HMI7HomeRunSel AND NOT #HMI8HomeRunSel AND NOT #HMI9HomeRunSel AND NOT #HMI10HomeRunSel) OR (NOT #HMI1HomeRunSel AND NOT #HMI2HomeRunSel AND NOT #HMI3HomeRunSel AND NOT #HMI4HomeRunSel AND NOT #HMI5HomeRunSel AND NOT #HMI6HomeRunSel AND NOT #HMI7HomeRunSel AND #HMI8HomeRunSel AND NOT #HMI9HomeRunSel AND NOT #HMI10HomeRunSel) OR (NOT #HMI1HomeRunSel AND NOT #HMI2HomeRunSel AND NOT #HMI3HomeRunSel AND NOT #HMI4HomeRunSel AND NOT #HMI5HomeRunSel AND NOT #HMI6HomeRunSel AND NOT #HMI7HomeRunSel AND NOT #HMI8HomeRunSel AND #HMI9HomeRunSel AND NOT #HMI10HomeRunSel) OR (NOT #HMI1HomeRunSel AND NOT #HMI2HomeRunSel AND NOT #HMI3HomeRunSel AND NOT #HMI4HomeRunSel AND NOT #HMI5HomeRunSel AND NOT #HMI6HomeRunSel AND NOT #HMI7HomeRunSel AND NOT #HMI8HomeRunSel AND NOT #HMI9HomeRunSel AND #HMI10HomeRunSel)) AND NOT #AutoSel;
   #IO_Modes.LModeSelector.HomeRunSel := #O_HomeRunSel;
END_REGION

REGION Network 99: **** 4.5 - Machine Status - Modes **** Reset activ HMI
   // Reset activ HMI
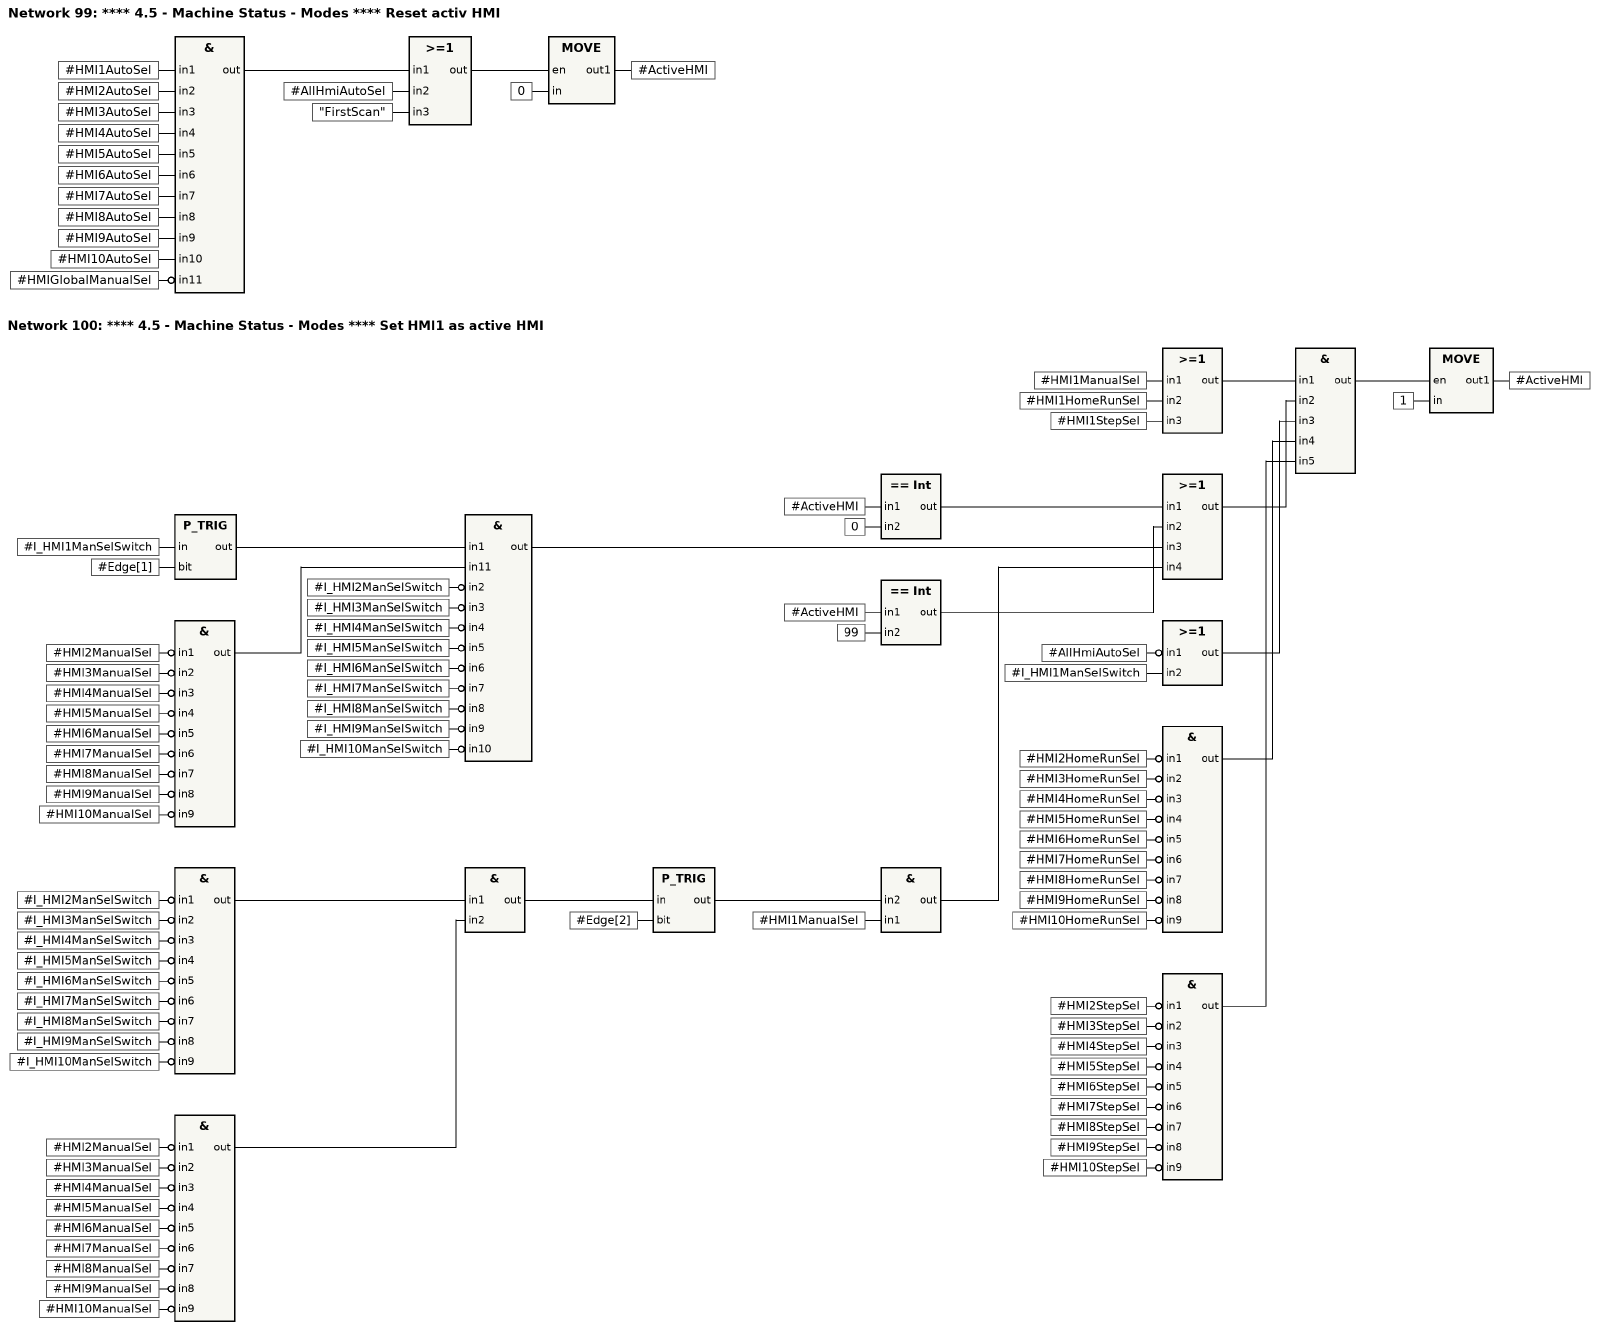
   IF (#HMI1AutoSel AND #HMI2AutoSel AND #HMI3AutoSel AND #HMI4AutoSel AND #HMI5AutoSel AND #HMI6AutoSel AND #HMI7AutoSel AND #HMI8AutoSel AND #HMI9AutoSel AND #HMI10AutoSel AND NOT #HMIGlobalManualSel) OR #AllHmiAutoSel OR "FirstScan" THEN
       #ActiveHMI := 0;
   END_IF;
END_REGION

REGION Network 100: **** 4.5 - Machine Status - Modes **** Set HMI1 as active HMI
   // Set HMI1 as active HMI
   #_w1 := #I_HMI1ManSelSwitch AND NOT #Edge[1];   // rising edge
   #Edge[1] := #I_HMI1ManSelSwitch;
   #_w2 := NOT #I_HMI2ManSelSwitch AND NOT #I_HMI3ManSelSwitch AND NOT #I_HMI4ManSelSwitch AND NOT #I_HMI5ManSelSwitch AND NOT #I_HMI6ManSelSwitch AND NOT #I_HMI7ManSelSwitch AND NOT #I_HMI8ManSelSwitch AND NOT #I_HMI9ManSelSwitch AND NOT #I_HMI10ManSelSwitch AND NOT #HMI2ManualSel AND NOT #HMI3ManualSel AND NOT #HMI4ManualSel AND NOT #HMI5ManualSel AND NOT #HMI6ManualSel AND NOT #HMI7ManualSel AND NOT #HMI8ManualSel AND NOT #HMI9ManualSel AND NOT #HMI10ManualSel;
   #_w3 := #_w2 AND NOT #Edge[2];   // rising edge
   #Edge[2] := #_w2;
   IF (#HMI1ManualSel OR #HMI1HomeRunSel OR #HMI1StepSel) AND ((#ActiveHMI = 0) OR (#ActiveHMI = 99) OR (#_w1 AND NOT #HMI2ManualSel AND NOT #HMI3ManualSel AND NOT #HMI4ManualSel AND NOT #HMI5ManualSel AND NOT #HMI6ManualSel AND NOT #HMI7ManualSel AND NOT #HMI8ManualSel AND NOT #HMI9ManualSel AND NOT #HMI10ManualSel AND NOT #I_HMI2ManSelSwitch AND NOT #I_HMI3ManSelSwitch AND NOT #I_HMI4ManSelSwitch AND NOT #I_HMI5ManSelSwitch AND NOT #I_HMI6ManSelSwitch AND NOT #I_HMI7ManSelSwitch AND NOT #I_HMI8ManSelSwitch AND NOT #I_HMI9ManSelSwitch AND NOT #I_HMI10ManSelSwitch) OR (#_w3 AND #HMI1ManualSel)) AND (NOT #AllHmiAutoSel OR #I_HMI1ManSelSwitch) AND NOT #HMI2HomeRunSel AND NOT #HMI3HomeRunSel AND NOT #HMI4HomeRunSel AND NOT #HMI5HomeRunSel AND NOT #HMI6HomeRunSel AND NOT #HMI7HomeRunSel AND NOT #HMI8HomeRunSel AND NOT #HMI9HomeRunSel AND NOT #HMI10HomeRunSel AND NOT #HMI2StepSel AND NOT #HMI3StepSel AND NOT #HMI4StepSel AND NOT #HMI5StepSel AND NOT #HMI6StepSel AND NOT #HMI7StepSel AND NOT #HMI8StepSel AND NOT #HMI9StepSel AND NOT #HMI10StepSel THEN
       #ActiveHMI := 1;
   END_IF;
END_REGION

REGION Network 101: **** 4.5 - Machine Status - Modes **** Set HMI2 as active HMI
   // Set HMI2 as active HMI
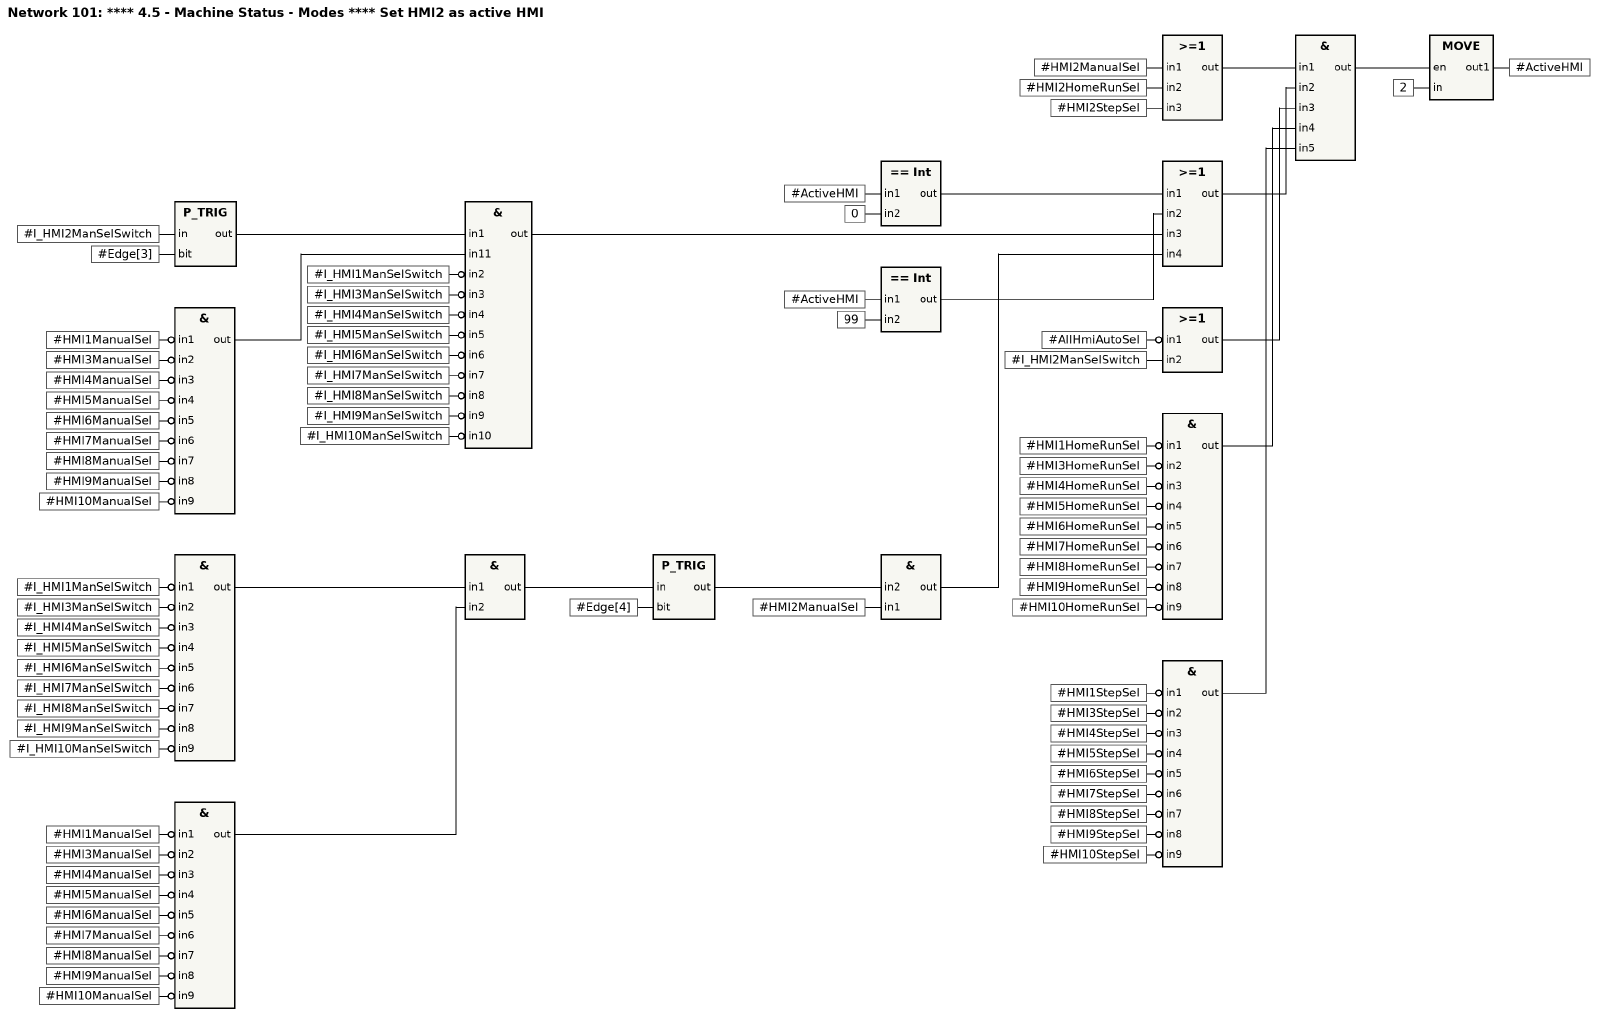
   #_w1 := #I_HMI2ManSelSwitch AND NOT #Edge[3];   // rising edge
   #Edge[3] := #I_HMI2ManSelSwitch;
   #_w2 := NOT #I_HMI1ManSelSwitch AND NOT #I_HMI3ManSelSwitch AND NOT #I_HMI4ManSelSwitch AND NOT #I_HMI5ManSelSwitch AND NOT #I_HMI6ManSelSwitch AND NOT #I_HMI7ManSelSwitch AND NOT #I_HMI8ManSelSwitch AND NOT #I_HMI9ManSelSwitch AND NOT #I_HMI10ManSelSwitch AND NOT #HMI1ManualSel AND NOT #HMI3ManualSel AND NOT #HMI4ManualSel AND NOT #HMI5ManualSel AND NOT #HMI6ManualSel AND NOT #HMI7ManualSel AND NOT #HMI8ManualSel AND NOT #HMI9ManualSel AND NOT #HMI10ManualSel;
   #_w3 := #_w2 AND NOT #Edge[4];   // rising edge
   #Edge[4] := #_w2;
   IF (#HMI2ManualSel OR #HMI2HomeRunSel OR #HMI2StepSel) AND ((#ActiveHMI = 0) OR (#ActiveHMI = 99) OR (#_w1 AND NOT #HMI1ManualSel AND NOT #HMI3ManualSel AND NOT #HMI4ManualSel AND NOT #HMI5ManualSel AND NOT #HMI6ManualSel AND NOT #HMI7ManualSel AND NOT #HMI8ManualSel AND NOT #HMI9ManualSel AND NOT #HMI10ManualSel AND NOT #I_HMI1ManSelSwitch AND NOT #I_HMI3ManSelSwitch AND NOT #I_HMI4ManSelSwitch AND NOT #I_HMI5ManSelSwitch AND NOT #I_HMI6ManSelSwitch AND NOT #I_HMI7ManSelSwitch AND NOT #I_HMI8ManSelSwitch AND NOT #I_HMI9ManSelSwitch AND NOT #I_HMI10ManSelSwitch) OR (#_w3 AND #HMI2ManualSel)) AND (NOT #AllHmiAutoSel OR #I_HMI2ManSelSwitch) AND NOT #HMI1HomeRunSel AND NOT #HMI3HomeRunSel AND NOT #HMI4HomeRunSel AND NOT #HMI5HomeRunSel AND NOT #HMI6HomeRunSel AND NOT #HMI7HomeRunSel AND NOT #HMI8HomeRunSel AND NOT #HMI9HomeRunSel AND NOT #HMI10HomeRunSel AND NOT #HMI1StepSel AND NOT #HMI3StepSel AND NOT #HMI4StepSel AND NOT #HMI5StepSel AND NOT #HMI6StepSel AND NOT #HMI7StepSel AND NOT #HMI8StepSel AND NOT #HMI9StepSel AND NOT #HMI10StepSel THEN
       #ActiveHMI := 2;
   END_IF;
END_REGION

REGION Network 102: **** 4.5 - Machine Status - Modes **** Set HMI3 as active HMI
   // Set HMI3 as active HMI
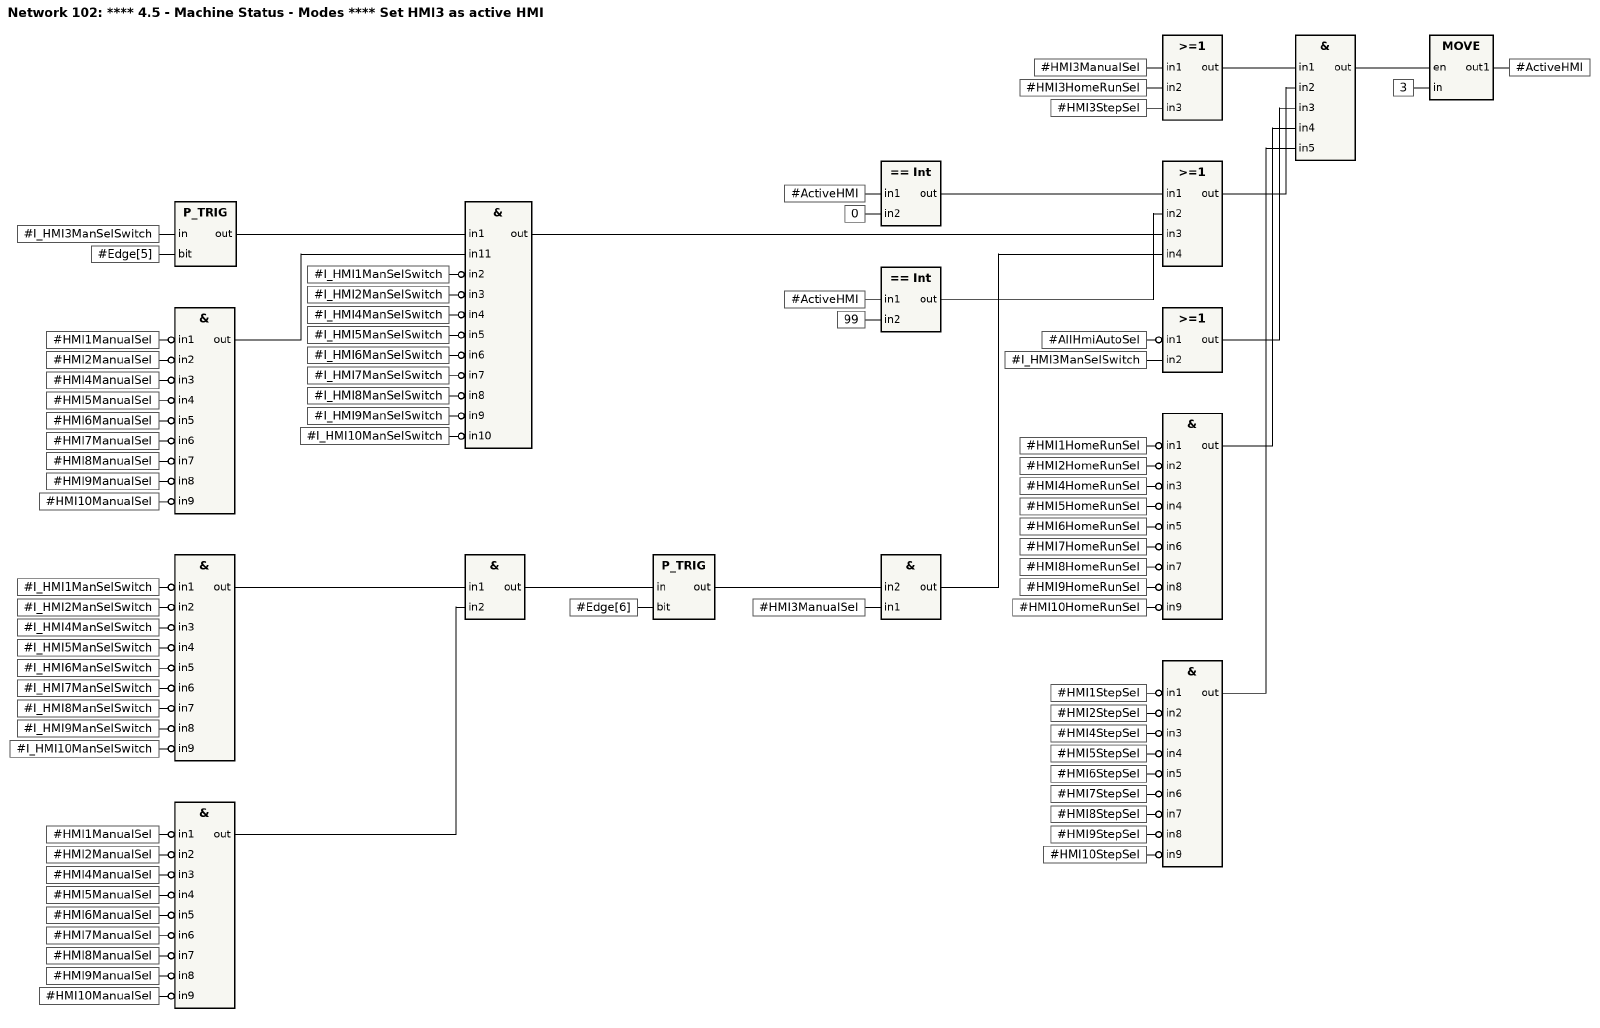
   #_w1 := #I_HMI3ManSelSwitch AND NOT #Edge[5];   // rising edge
   #Edge[5] := #I_HMI3ManSelSwitch;
   #_w2 := NOT #I_HMI1ManSelSwitch AND NOT #I_HMI2ManSelSwitch AND NOT #I_HMI4ManSelSwitch AND NOT #I_HMI5ManSelSwitch AND NOT #I_HMI6ManSelSwitch AND NOT #I_HMI7ManSelSwitch AND NOT #I_HMI8ManSelSwitch AND NOT #I_HMI9ManSelSwitch AND NOT #I_HMI10ManSelSwitch AND NOT #HMI1ManualSel AND NOT #HMI2ManualSel AND NOT #HMI4ManualSel AND NOT #HMI5ManualSel AND NOT #HMI6ManualSel AND NOT #HMI7ManualSel AND NOT #HMI8ManualSel AND NOT #HMI9ManualSel AND NOT #HMI10ManualSel;
   #_w3 := #_w2 AND NOT #Edge[6];   // rising edge
   #Edge[6] := #_w2;
   IF (#HMI3ManualSel OR #HMI3HomeRunSel OR #HMI3StepSel) AND ((#ActiveHMI = 0) OR (#ActiveHMI = 99) OR (#_w1 AND NOT #HMI1ManualSel AND NOT #HMI2ManualSel AND NOT #HMI4ManualSel AND NOT #HMI5ManualSel AND NOT #HMI6ManualSel AND NOT #HMI7ManualSel AND NOT #HMI8ManualSel AND NOT #HMI9ManualSel AND NOT #HMI10ManualSel AND NOT #I_HMI1ManSelSwitch AND NOT #I_HMI2ManSelSwitch AND NOT #I_HMI4ManSelSwitch AND NOT #I_HMI5ManSelSwitch AND NOT #I_HMI6ManSelSwitch AND NOT #I_HMI7ManSelSwitch AND NOT #I_HMI8ManSelSwitch AND NOT #I_HMI9ManSelSwitch AND NOT #I_HMI10ManSelSwitch) OR (#_w3 AND #HMI3ManualSel)) AND (NOT #AllHmiAutoSel OR #I_HMI3ManSelSwitch) AND NOT #HMI1HomeRunSel AND NOT #HMI2HomeRunSel AND NOT #HMI4HomeRunSel AND NOT #HMI5HomeRunSel AND NOT #HMI6HomeRunSel AND NOT #HMI7HomeRunSel AND NOT #HMI8HomeRunSel AND NOT #HMI9HomeRunSel AND NOT #HMI10HomeRunSel AND NOT #HMI1StepSel AND NOT #HMI2StepSel AND NOT #HMI4StepSel AND NOT #HMI5StepSel AND NOT #HMI6StepSel AND NOT #HMI7StepSel AND NOT #HMI8StepSel AND NOT #HMI9StepSel AND NOT #HMI10StepSel THEN
       #ActiveHMI := 3;
   END_IF;
END_REGION

REGION Network 103: **** 4.5 - Machine Status - Modes **** Set HMI4 as active HMI
   // Set HMI4 as active HMI
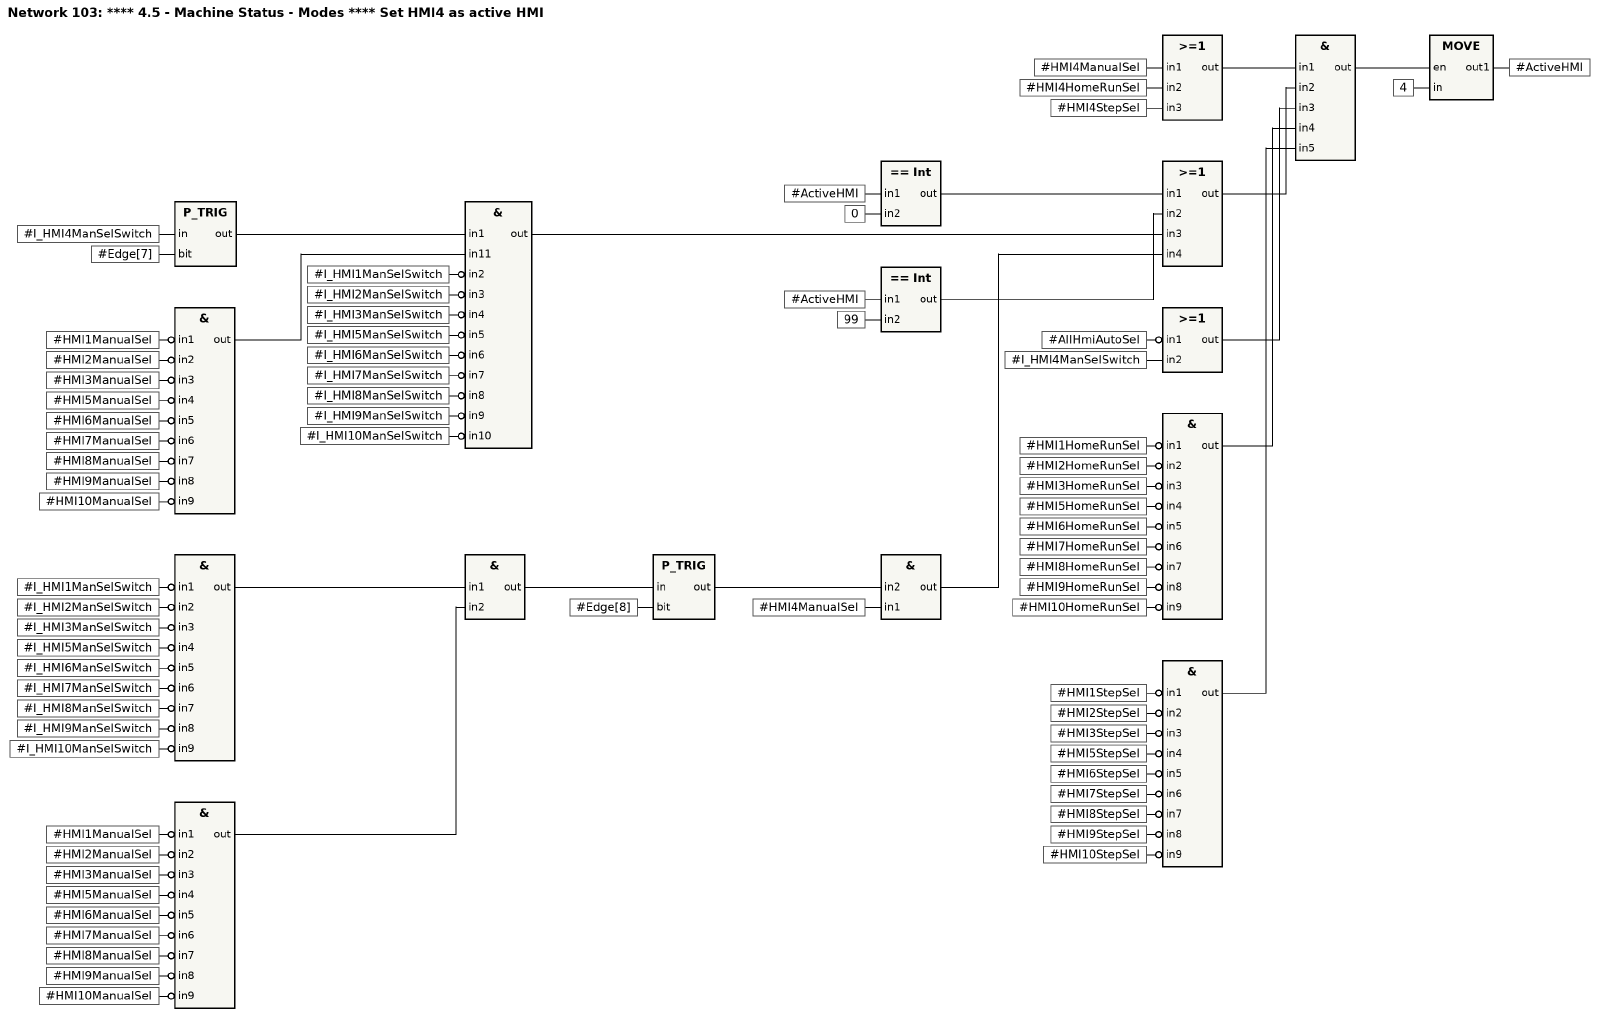
   #_w1 := #I_HMI4ManSelSwitch AND NOT #Edge[7];   // rising edge
   #Edge[7] := #I_HMI4ManSelSwitch;
   #_w2 := NOT #I_HMI1ManSelSwitch AND NOT #I_HMI2ManSelSwitch AND NOT #I_HMI3ManSelSwitch AND NOT #I_HMI5ManSelSwitch AND NOT #I_HMI6ManSelSwitch AND NOT #I_HMI7ManSelSwitch AND NOT #I_HMI8ManSelSwitch AND NOT #I_HMI9ManSelSwitch AND NOT #I_HMI10ManSelSwitch AND NOT #HMI1ManualSel AND NOT #HMI2ManualSel AND NOT #HMI3ManualSel AND NOT #HMI5ManualSel AND NOT #HMI6ManualSel AND NOT #HMI7ManualSel AND NOT #HMI8ManualSel AND NOT #HMI9ManualSel AND NOT #HMI10ManualSel;
   #_w3 := #_w2 AND NOT #Edge[8];   // rising edge
   #Edge[8] := #_w2;
   IF (#HMI4ManualSel OR #HMI4HomeRunSel OR #HMI4StepSel) AND ((#ActiveHMI = 0) OR (#ActiveHMI = 99) OR (#_w1 AND NOT #HMI1ManualSel AND NOT #HMI2ManualSel AND NOT #HMI3ManualSel AND NOT #HMI5ManualSel AND NOT #HMI6ManualSel AND NOT #HMI7ManualSel AND NOT #HMI8ManualSel AND NOT #HMI9ManualSel AND NOT #HMI10ManualSel AND NOT #I_HMI1ManSelSwitch AND NOT #I_HMI2ManSelSwitch AND NOT #I_HMI3ManSelSwitch AND NOT #I_HMI5ManSelSwitch AND NOT #I_HMI6ManSelSwitch AND NOT #I_HMI7ManSelSwitch AND NOT #I_HMI8ManSelSwitch AND NOT #I_HMI9ManSelSwitch AND NOT #I_HMI10ManSelSwitch) OR (#_w3 AND #HMI4ManualSel)) AND (NOT #AllHmiAutoSel OR #I_HMI4ManSelSwitch) AND NOT #HMI1HomeRunSel AND NOT #HMI2HomeRunSel AND NOT #HMI3HomeRunSel AND NOT #HMI5HomeRunSel AND NOT #HMI6HomeRunSel AND NOT #HMI7HomeRunSel AND NOT #HMI8HomeRunSel AND NOT #HMI9HomeRunSel AND NOT #HMI10HomeRunSel AND NOT #HMI1StepSel AND NOT #HMI2StepSel AND NOT #HMI3StepSel AND NOT #HMI5StepSel AND NOT #HMI6StepSel AND NOT #HMI7StepSel AND NOT #HMI8StepSel AND NOT #HMI9StepSel AND NOT #HMI10StepSel THEN
       #ActiveHMI := 4;
   END_IF;
END_REGION

REGION Network 104: **** 4.5 - Machine Status - Modes **** Set HMI5 as active HMI
   // Set HMI5 as active HMI
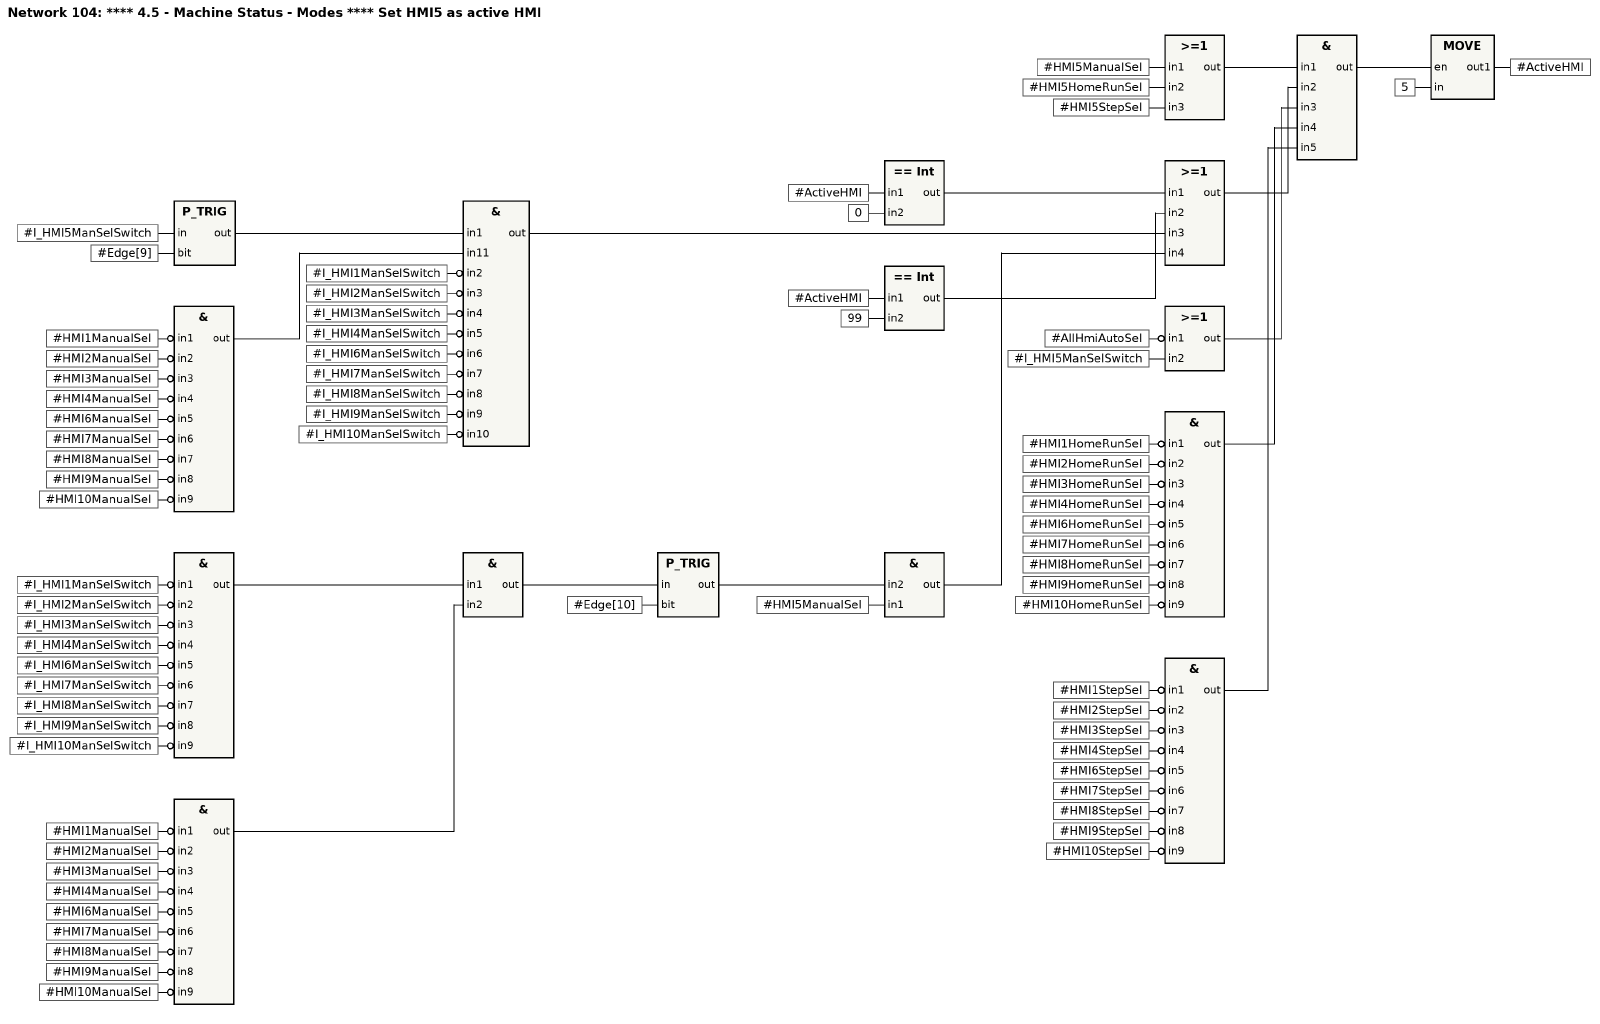
   #_w1 := #I_HMI5ManSelSwitch AND NOT #Edge[9];   // rising edge
   #Edge[9] := #I_HMI5ManSelSwitch;
   #_w2 := NOT #I_HMI1ManSelSwitch AND NOT #I_HMI2ManSelSwitch AND NOT #I_HMI3ManSelSwitch AND NOT #I_HMI4ManSelSwitch AND NOT #I_HMI6ManSelSwitch AND NOT #I_HMI7ManSelSwitch AND NOT #I_HMI8ManSelSwitch AND NOT #I_HMI9ManSelSwitch AND NOT #I_HMI10ManSelSwitch AND NOT #HMI1ManualSel AND NOT #HMI2ManualSel AND NOT #HMI3ManualSel AND NOT #HMI4ManualSel AND NOT #HMI6ManualSel AND NOT #HMI7ManualSel AND NOT #HMI8ManualSel AND NOT #HMI9ManualSel AND NOT #HMI10ManualSel;
   #_w3 := #_w2 AND NOT #Edge[10];   // rising edge
   #Edge[10] := #_w2;
   IF (#HMI5ManualSel OR #HMI5HomeRunSel OR #HMI5StepSel) AND ((#ActiveHMI = 0) OR (#ActiveHMI = 99) OR (#_w1 AND NOT #HMI1ManualSel AND NOT #HMI2ManualSel AND NOT #HMI3ManualSel AND NOT #HMI4ManualSel AND NOT #HMI6ManualSel AND NOT #HMI7ManualSel AND NOT #HMI8ManualSel AND NOT #HMI9ManualSel AND NOT #HMI10ManualSel AND NOT #I_HMI1ManSelSwitch AND NOT #I_HMI2ManSelSwitch AND NOT #I_HMI3ManSelSwitch AND NOT #I_HMI4ManSelSwitch AND NOT #I_HMI6ManSelSwitch AND NOT #I_HMI7ManSelSwitch AND NOT #I_HMI8ManSelSwitch AND NOT #I_HMI9ManSelSwitch AND NOT #I_HMI10ManSelSwitch) OR (#_w3 AND #HMI5ManualSel)) AND (NOT #AllHmiAutoSel OR #I_HMI5ManSelSwitch) AND NOT #HMI1HomeRunSel AND NOT #HMI2HomeRunSel AND NOT #HMI3HomeRunSel AND NOT #HMI4HomeRunSel AND NOT #HMI6HomeRunSel AND NOT #HMI7HomeRunSel AND NOT #HMI8HomeRunSel AND NOT #HMI9HomeRunSel AND NOT #HMI10HomeRunSel AND NOT #HMI1StepSel AND NOT #HMI2StepSel AND NOT #HMI3StepSel AND NOT #HMI4StepSel AND NOT #HMI6StepSel AND NOT #HMI7StepSel AND NOT #HMI8StepSel AND NOT #HMI9StepSel AND NOT #HMI10StepSel THEN
       #ActiveHMI := 5;
   END_IF;
END_REGION

REGION Network 105: **** 4.5 - Machine Status - Modes **** Set HMI6 as active HMI
   // Set HMI6 as active HMI
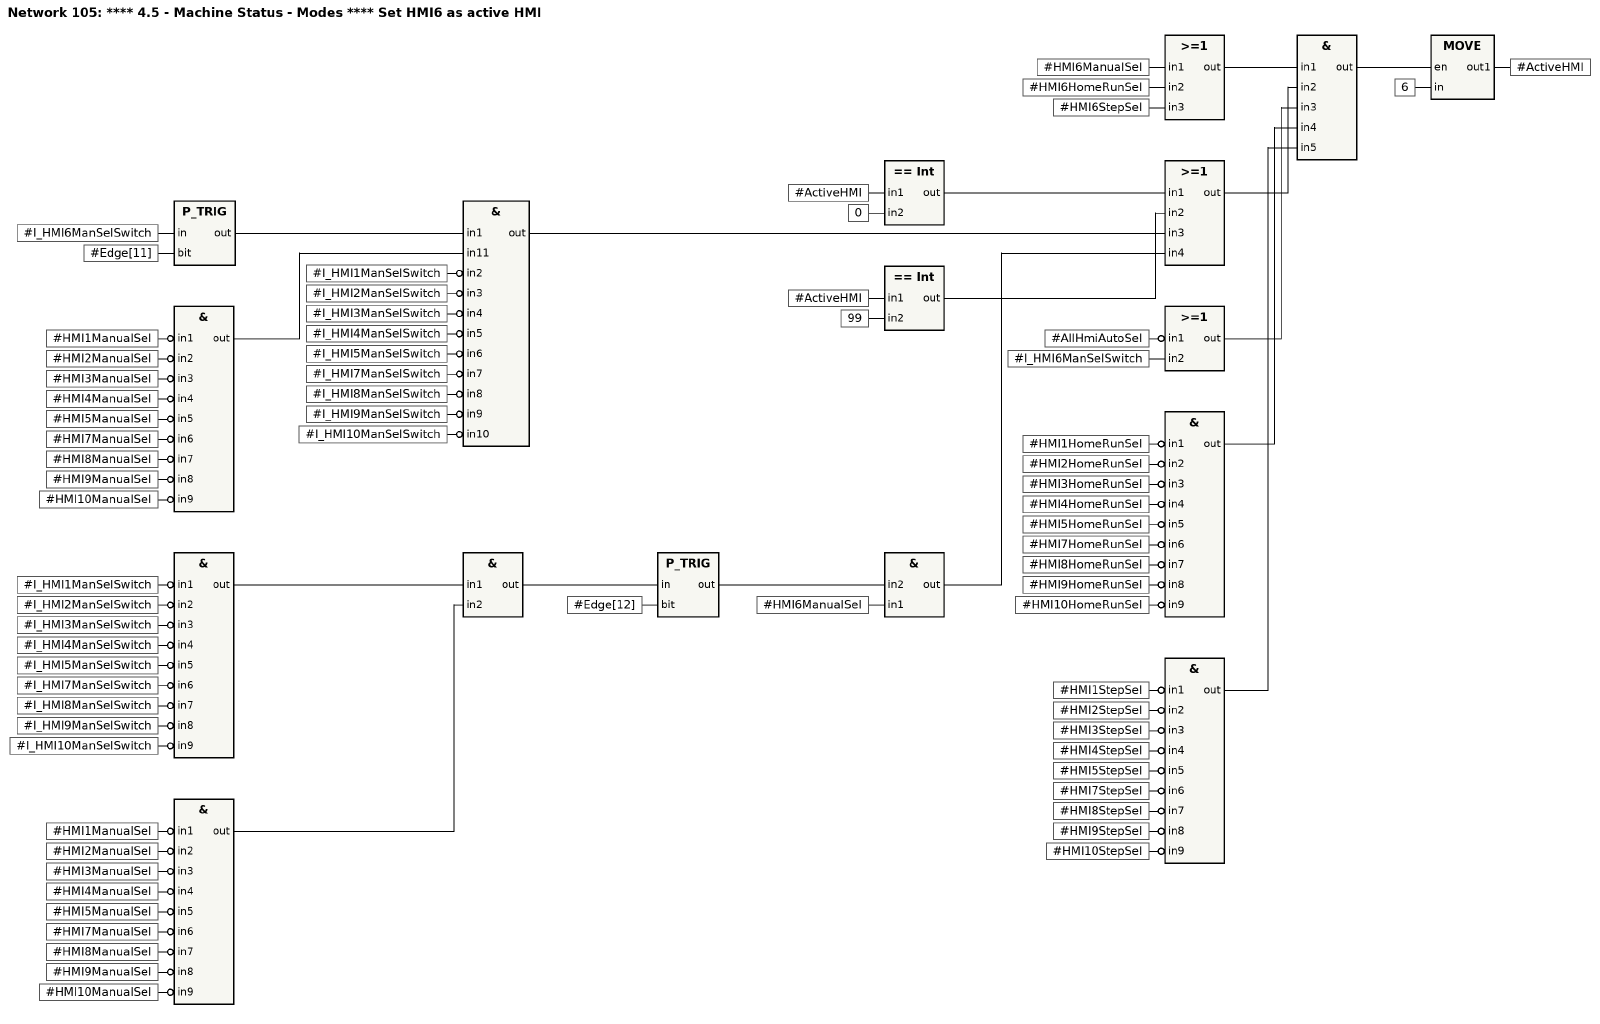
   #_w1 := #I_HMI6ManSelSwitch AND NOT #Edge[11];   // rising edge
   #Edge[11] := #I_HMI6ManSelSwitch;
   #_w2 := NOT #I_HMI1ManSelSwitch AND NOT #I_HMI2ManSelSwitch AND NOT #I_HMI3ManSelSwitch AND NOT #I_HMI4ManSelSwitch AND NOT #I_HMI5ManSelSwitch AND NOT #I_HMI7ManSelSwitch AND NOT #I_HMI8ManSelSwitch AND NOT #I_HMI9ManSelSwitch AND NOT #I_HMI10ManSelSwitch AND NOT #HMI1ManualSel AND NOT #HMI2ManualSel AND NOT #HMI3ManualSel AND NOT #HMI4ManualSel AND NOT #HMI5ManualSel AND NOT #HMI7ManualSel AND NOT #HMI8ManualSel AND NOT #HMI9ManualSel AND NOT #HMI10ManualSel;
   #_w3 := #_w2 AND NOT #Edge[12];   // rising edge
   #Edge[12] := #_w2;
   IF (#HMI6ManualSel OR #HMI6HomeRunSel OR #HMI6StepSel) AND ((#ActiveHMI = 0) OR (#ActiveHMI = 99) OR (#_w1 AND NOT #HMI1ManualSel AND NOT #HMI2ManualSel AND NOT #HMI3ManualSel AND NOT #HMI4ManualSel AND NOT #HMI5ManualSel AND NOT #HMI7ManualSel AND NOT #HMI8ManualSel AND NOT #HMI9ManualSel AND NOT #HMI10ManualSel AND NOT #I_HMI1ManSelSwitch AND NOT #I_HMI2ManSelSwitch AND NOT #I_HMI3ManSelSwitch AND NOT #I_HMI4ManSelSwitch AND NOT #I_HMI5ManSelSwitch AND NOT #I_HMI7ManSelSwitch AND NOT #I_HMI8ManSelSwitch AND NOT #I_HMI9ManSelSwitch AND NOT #I_HMI10ManSelSwitch) OR (#_w3 AND #HMI6ManualSel)) AND (NOT #AllHmiAutoSel OR #I_HMI6ManSelSwitch) AND NOT #HMI1HomeRunSel AND NOT #HMI2HomeRunSel AND NOT #HMI3HomeRunSel AND NOT #HMI4HomeRunSel AND NOT #HMI5HomeRunSel AND NOT #HMI7HomeRunSel AND NOT #HMI8HomeRunSel AND NOT #HMI9HomeRunSel AND NOT #HMI10HomeRunSel AND NOT #HMI1StepSel AND NOT #HMI2StepSel AND NOT #HMI3StepSel AND NOT #HMI4StepSel AND NOT #HMI5StepSel AND NOT #HMI7StepSel AND NOT #HMI8StepSel AND NOT #HMI9StepSel AND NOT #HMI10StepSel THEN
       #ActiveHMI := 6;
   END_IF;
END_REGION

REGION Network 106: **** 4.5 - Machine Status - Modes **** Set HMI7 as active HMI
   // Set HMI7 as active HMI
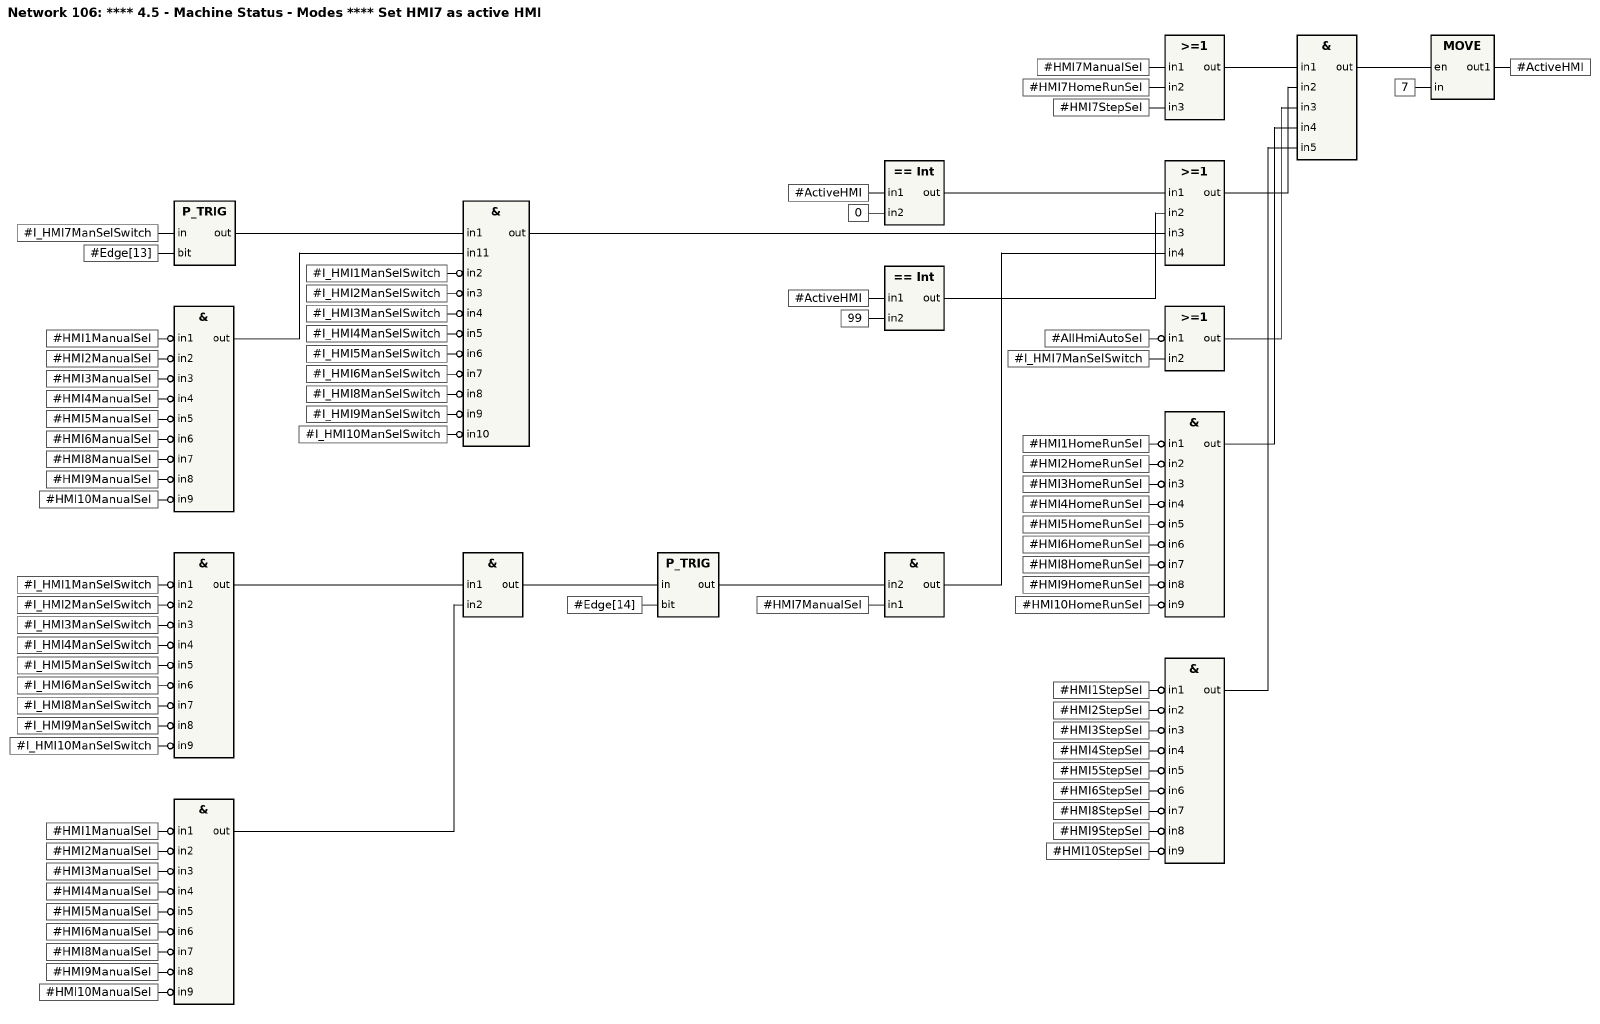
   #_w1 := #I_HMI7ManSelSwitch AND NOT #Edge[13];   // rising edge
   #Edge[13] := #I_HMI7ManSelSwitch;
   #_w2 := NOT #I_HMI1ManSelSwitch AND NOT #I_HMI2ManSelSwitch AND NOT #I_HMI3ManSelSwitch AND NOT #I_HMI4ManSelSwitch AND NOT #I_HMI5ManSelSwitch AND NOT #I_HMI6ManSelSwitch AND NOT #I_HMI8ManSelSwitch AND NOT #I_HMI9ManSelSwitch AND NOT #I_HMI10ManSelSwitch AND NOT #HMI1ManualSel AND NOT #HMI2ManualSel AND NOT #HMI3ManualSel AND NOT #HMI4ManualSel AND NOT #HMI5ManualSel AND NOT #HMI6ManualSel AND NOT #HMI8ManualSel AND NOT #HMI9ManualSel AND NOT #HMI10ManualSel;
   #_w3 := #_w2 AND NOT #Edge[14];   // rising edge
   #Edge[14] := #_w2;
   IF (#HMI7ManualSel OR #HMI7HomeRunSel OR #HMI7StepSel) AND ((#ActiveHMI = 0) OR (#ActiveHMI = 99) OR (#_w1 AND NOT #HMI1ManualSel AND NOT #HMI2ManualSel AND NOT #HMI3ManualSel AND NOT #HMI4ManualSel AND NOT #HMI5ManualSel AND NOT #HMI6ManualSel AND NOT #HMI8ManualSel AND NOT #HMI9ManualSel AND NOT #HMI10ManualSel AND NOT #I_HMI1ManSelSwitch AND NOT #I_HMI2ManSelSwitch AND NOT #I_HMI3ManSelSwitch AND NOT #I_HMI4ManSelSwitch AND NOT #I_HMI5ManSelSwitch AND NOT #I_HMI6ManSelSwitch AND NOT #I_HMI8ManSelSwitch AND NOT #I_HMI9ManSelSwitch AND NOT #I_HMI10ManSelSwitch) OR (#_w3 AND #HMI7ManualSel)) AND (NOT #AllHmiAutoSel OR #I_HMI7ManSelSwitch) AND NOT #HMI1HomeRunSel AND NOT #HMI2HomeRunSel AND NOT #HMI3HomeRunSel AND NOT #HMI4HomeRunSel AND NOT #HMI5HomeRunSel AND NOT #HMI6HomeRunSel AND NOT #HMI8HomeRunSel AND NOT #HMI9HomeRunSel AND NOT #HMI10HomeRunSel AND NOT #HMI1StepSel AND NOT #HMI2StepSel AND NOT #HMI3StepSel AND NOT #HMI4StepSel AND NOT #HMI5StepSel AND NOT #HMI6StepSel AND NOT #HMI8StepSel AND NOT #HMI9StepSel AND NOT #HMI10StepSel THEN
       #ActiveHMI := 7;
   END_IF;
END_REGION

REGION Network 107: **** 4.5 - Machine Status - Modes **** Set HMI8 as active HMI
   // Set HMI8 as active HMI
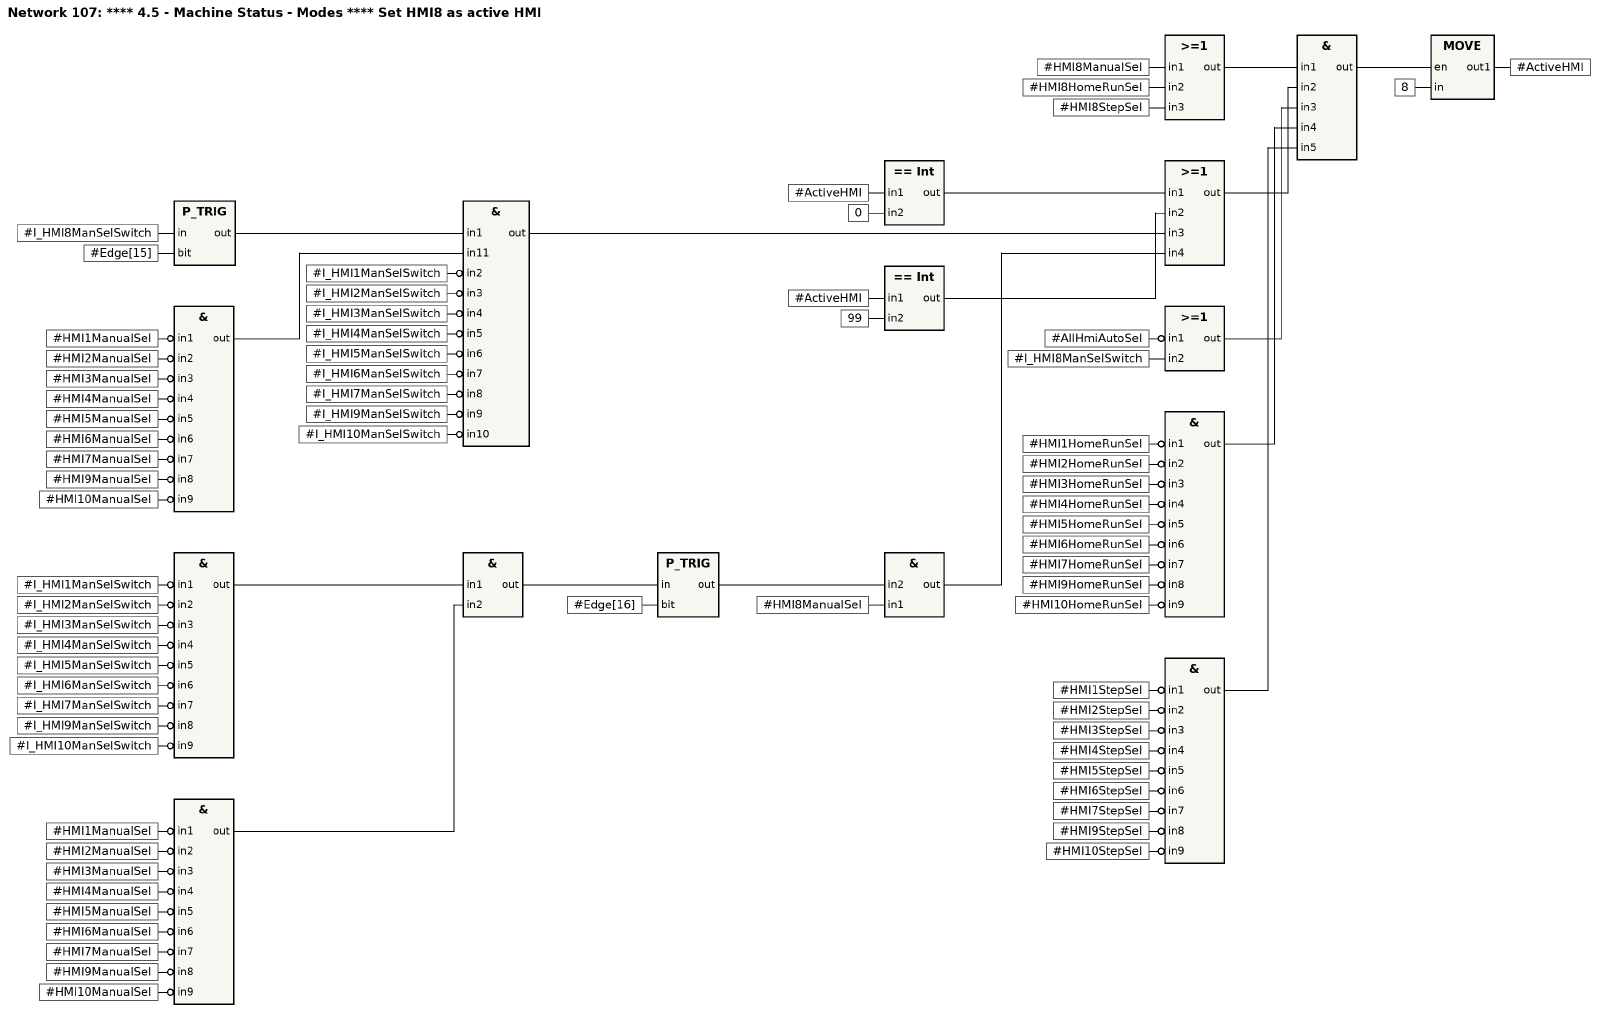
   #_w1 := #I_HMI8ManSelSwitch AND NOT #Edge[15];   // rising edge
   #Edge[15] := #I_HMI8ManSelSwitch;
   #_w2 := NOT #I_HMI1ManSelSwitch AND NOT #I_HMI2ManSelSwitch AND NOT #I_HMI3ManSelSwitch AND NOT #I_HMI4ManSelSwitch AND NOT #I_HMI5ManSelSwitch AND NOT #I_HMI6ManSelSwitch AND NOT #I_HMI7ManSelSwitch AND NOT #I_HMI9ManSelSwitch AND NOT #I_HMI10ManSelSwitch AND NOT #HMI1ManualSel AND NOT #HMI2ManualSel AND NOT #HMI3ManualSel AND NOT #HMI4ManualSel AND NOT #HMI5ManualSel AND NOT #HMI6ManualSel AND NOT #HMI7ManualSel AND NOT #HMI9ManualSel AND NOT #HMI10ManualSel;
   #_w3 := #_w2 AND NOT #Edge[16];   // rising edge
   #Edge[16] := #_w2;
   IF (#HMI8ManualSel OR #HMI8HomeRunSel OR #HMI8StepSel) AND ((#ActiveHMI = 0) OR (#ActiveHMI = 99) OR (#_w1 AND NOT #HMI1ManualSel AND NOT #HMI2ManualSel AND NOT #HMI3ManualSel AND NOT #HMI4ManualSel AND NOT #HMI5ManualSel AND NOT #HMI6ManualSel AND NOT #HMI7ManualSel AND NOT #HMI9ManualSel AND NOT #HMI10ManualSel AND NOT #I_HMI1ManSelSwitch AND NOT #I_HMI2ManSelSwitch AND NOT #I_HMI3ManSelSwitch AND NOT #I_HMI4ManSelSwitch AND NOT #I_HMI5ManSelSwitch AND NOT #I_HMI6ManSelSwitch AND NOT #I_HMI7ManSelSwitch AND NOT #I_HMI9ManSelSwitch AND NOT #I_HMI10ManSelSwitch) OR (#_w3 AND #HMI8ManualSel)) AND (NOT #AllHmiAutoSel OR #I_HMI8ManSelSwitch) AND NOT #HMI1HomeRunSel AND NOT #HMI2HomeRunSel AND NOT #HMI3HomeRunSel AND NOT #HMI4HomeRunSel AND NOT #HMI5HomeRunSel AND NOT #HMI6HomeRunSel AND NOT #HMI7HomeRunSel AND NOT #HMI9HomeRunSel AND NOT #HMI10HomeRunSel AND NOT #HMI1StepSel AND NOT #HMI2StepSel AND NOT #HMI3StepSel AND NOT #HMI4StepSel AND NOT #HMI5StepSel AND NOT #HMI6StepSel AND NOT #HMI7StepSel AND NOT #HMI9StepSel AND NOT #HMI10StepSel THEN
       #ActiveHMI := 8;
   END_IF;
END_REGION

REGION Network 108: **** 4.5 - Machine Status - Modes **** Set HMI9 as active HMI
   // Set HMI9 as active HMI
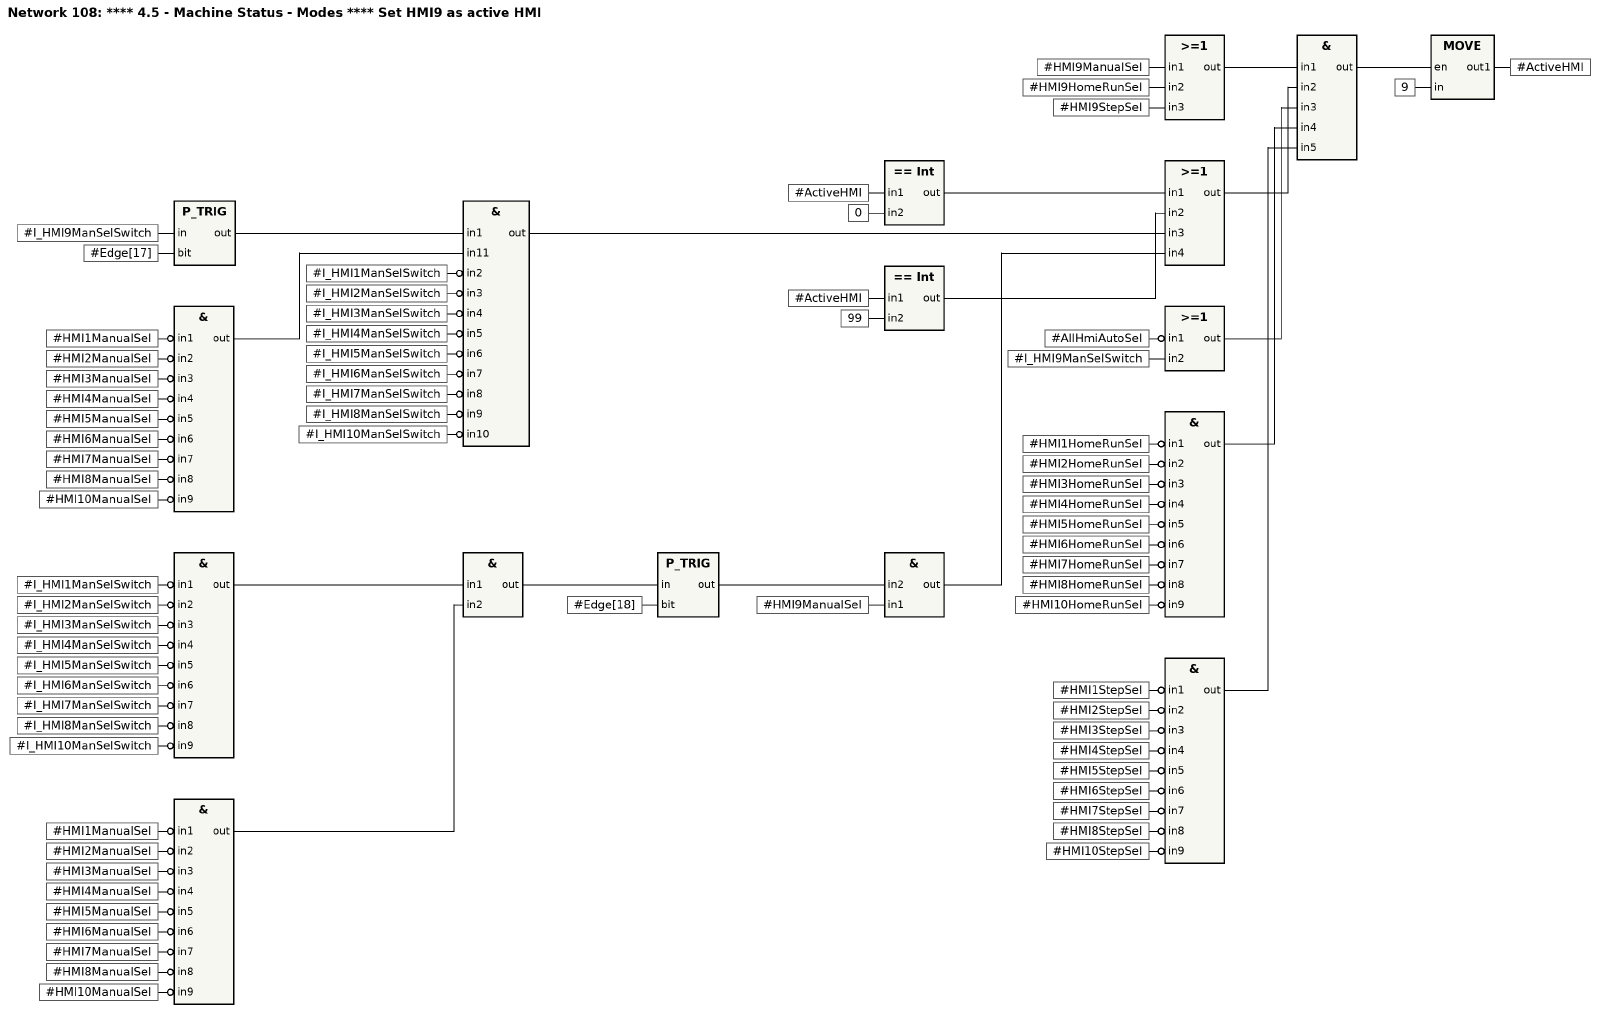
   #_w1 := #I_HMI9ManSelSwitch AND NOT #Edge[17];   // rising edge
   #Edge[17] := #I_HMI9ManSelSwitch;
   #_w2 := NOT #I_HMI1ManSelSwitch AND NOT #I_HMI2ManSelSwitch AND NOT #I_HMI3ManSelSwitch AND NOT #I_HMI4ManSelSwitch AND NOT #I_HMI5ManSelSwitch AND NOT #I_HMI6ManSelSwitch AND NOT #I_HMI7ManSelSwitch AND NOT #I_HMI8ManSelSwitch AND NOT #I_HMI10ManSelSwitch AND NOT #HMI1ManualSel AND NOT #HMI2ManualSel AND NOT #HMI3ManualSel AND NOT #HMI4ManualSel AND NOT #HMI5ManualSel AND NOT #HMI6ManualSel AND NOT #HMI7ManualSel AND NOT #HMI8ManualSel AND NOT #HMI10ManualSel;
   #_w3 := #_w2 AND NOT #Edge[18];   // rising edge
   #Edge[18] := #_w2;
   IF (#HMI9ManualSel OR #HMI9HomeRunSel OR #HMI9StepSel) AND ((#ActiveHMI = 0) OR (#ActiveHMI = 99) OR (#_w1 AND NOT #HMI1ManualSel AND NOT #HMI2ManualSel AND NOT #HMI3ManualSel AND NOT #HMI4ManualSel AND NOT #HMI5ManualSel AND NOT #HMI6ManualSel AND NOT #HMI7ManualSel AND NOT #HMI8ManualSel AND NOT #HMI10ManualSel AND NOT #I_HMI1ManSelSwitch AND NOT #I_HMI2ManSelSwitch AND NOT #I_HMI3ManSelSwitch AND NOT #I_HMI4ManSelSwitch AND NOT #I_HMI5ManSelSwitch AND NOT #I_HMI6ManSelSwitch AND NOT #I_HMI7ManSelSwitch AND NOT #I_HMI8ManSelSwitch AND NOT #I_HMI10ManSelSwitch) OR (#_w3 AND #HMI9ManualSel)) AND (NOT #AllHmiAutoSel OR #I_HMI9ManSelSwitch) AND NOT #HMI1HomeRunSel AND NOT #HMI2HomeRunSel AND NOT #HMI3HomeRunSel AND NOT #HMI4HomeRunSel AND NOT #HMI5HomeRunSel AND NOT #HMI6HomeRunSel AND NOT #HMI7HomeRunSel AND NOT #HMI8HomeRunSel AND NOT #HMI10HomeRunSel AND NOT #HMI1StepSel AND NOT #HMI2StepSel AND NOT #HMI3StepSel AND NOT #HMI4StepSel AND NOT #HMI5StepSel AND NOT #HMI6StepSel AND NOT #HMI7StepSel AND NOT #HMI8StepSel AND NOT #HMI10StepSel THEN
       #ActiveHMI := 9;
   END_IF;
END_REGION

REGION Network 109: **** 4.5 - Machine Status - Modes **** Set HMI10 as active HMI
   // Set HMI10 as active HMI
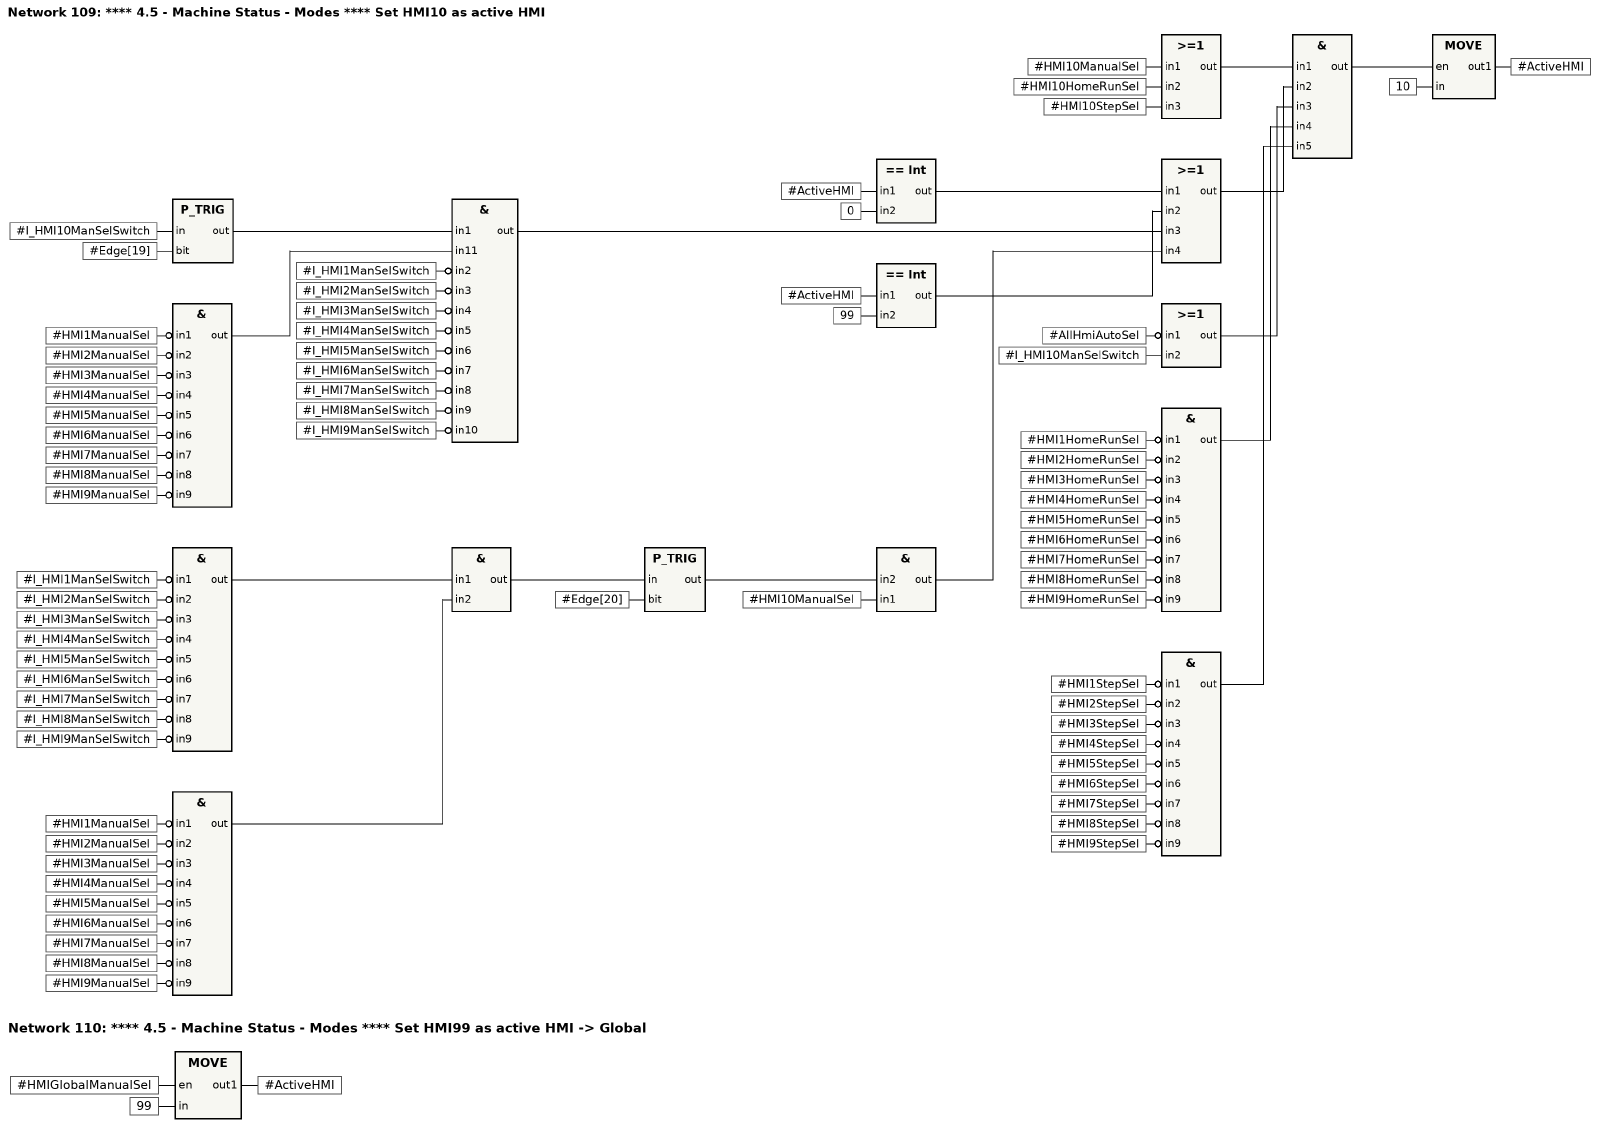
   #_w1 := #I_HMI10ManSelSwitch AND NOT #Edge[19];   // rising edge
   #Edge[19] := #I_HMI10ManSelSwitch;
   #_w2 := NOT #I_HMI1ManSelSwitch AND NOT #I_HMI2ManSelSwitch AND NOT #I_HMI3ManSelSwitch AND NOT #I_HMI4ManSelSwitch AND NOT #I_HMI5ManSelSwitch AND NOT #I_HMI6ManSelSwitch AND NOT #I_HMI7ManSelSwitch AND NOT #I_HMI8ManSelSwitch AND NOT #I_HMI9ManSelSwitch AND NOT #HMI1ManualSel AND NOT #HMI2ManualSel AND NOT #HMI3ManualSel AND NOT #HMI4ManualSel AND NOT #HMI5ManualSel AND NOT #HMI6ManualSel AND NOT #HMI7ManualSel AND NOT #HMI8ManualSel AND NOT #HMI9ManualSel;
   #_w3 := #_w2 AND NOT #Edge[20];   // rising edge
   #Edge[20] := #_w2;
   IF (#HMI10ManualSel OR #HMI10HomeRunSel OR #HMI10StepSel) AND ((#ActiveHMI = 0) OR (#ActiveHMI = 99) OR (#_w1 AND NOT #HMI1ManualSel AND NOT #HMI2ManualSel AND NOT #HMI3ManualSel AND NOT #HMI4ManualSel AND NOT #HMI5ManualSel AND NOT #HMI6ManualSel AND NOT #HMI7ManualSel AND NOT #HMI8ManualSel AND NOT #HMI9ManualSel AND NOT #I_HMI1ManSelSwitch AND NOT #I_HMI2ManSelSwitch AND NOT #I_HMI3ManSelSwitch AND NOT #I_HMI4ManSelSwitch AND NOT #I_HMI5ManSelSwitch AND NOT #I_HMI6ManSelSwitch AND NOT #I_HMI7ManSelSwitch AND NOT #I_HMI8ManSelSwitch AND NOT #I_HMI9ManSelSwitch) OR (#_w3 AND #HMI10ManualSel)) AND (NOT #AllHmiAutoSel OR #I_HMI10ManSelSwitch) AND NOT #HMI1HomeRunSel AND NOT #HMI2HomeRunSel AND NOT #HMI3HomeRunSel AND NOT #HMI4HomeRunSel AND NOT #HMI5HomeRunSel AND NOT #HMI6HomeRunSel AND NOT #HMI7HomeRunSel AND NOT #HMI8HomeRunSel AND NOT #HMI9HomeRunSel AND NOT #HMI1StepSel AND NOT #HMI2StepSel AND NOT #HMI3StepSel AND NOT #HMI4StepSel AND NOT #HMI5StepSel AND NOT #HMI6StepSel AND NOT #HMI7StepSel AND NOT #HMI8StepSel AND NOT #HMI9StepSel THEN
       #ActiveHMI := 10;
   END_IF;
END_REGION

REGION Network 110: **** 4.5 - Machine Status - Modes **** Set HMI99 as active HMI -> Global
   IF #HMIGlobalManualSel THEN #ActiveHMI := 99; END_IF;
END_REGION

REGION Network 111: **** 4.5 - Machine Status - Modes **** Set Manual selected if one of the HMI is active
   // Set Manual selected if one of the HMI is active
